LIN {X 0,Y 305.425,Z 148.042,A -85,B 0,C 180,E1 -16066.344,E2 -16066.344} C_VEL
LIN {X 0,Y 305.415,Z 148.066,A -85,B 0,C 180,E1 -16069.885,E2 -16069.885} C_VEL
LIN {X 0,Y 305.467,Z 148.054,A -85,B 0,C 180,E1 -16073.636,E2 -16073.636} C_VEL
LIN {X 0,Y 305.47,Z 148.051,A -85,B 0,C 180,E1 -16076.483,E2 -16076.483} C_VEL
LIN {X 0,Y 305.436,Z 148.065,A -85,B 0,C 180,E1 -16079.587,E2 -16079.587} C_VEL
LIN {X 0,Y 305.456,Z 148.059,A -85,B 0,C 180,E1 -16082.602,E2 -16082.602} C_VEL
LIN {X 0,Y 305.461,Z 148.064,A -85,B 0,C 180,E1 -16085.534,E2 -16085.534} C_VEL
LIN {X 0,Y 305.504,Z 148.057,A -85,B 0,C 180,E1 -16089.813,E2 -16089.813} C_VEL
LIN {X 0,Y 305.56,Z 148.153,A -85,B 0,C 180,E1 -16092.669,E2 -16092.669} C_VEL
LIN {X 0,Y 306.725,Z 151.141,A -85,B 0,C 180,E1 -16092.931,E2 -16092.931} C_VEL
LIN {X 0,Y 311.745,Z 160.729,A -85,B 0,C 180,E1 -16093.747,E2 -16093.747} C_VEL
LIN {X 0,Y 320.601,Z 180.222,A -85,B 0,C 180,E1 -16095.182,E2 -16095.182} C_VEL
LIN {X 0,Y 326.991,Z 195.626,A -85,B 0,C 180,E1 -16096.196,E2 -16096.196} C_VEL
LIN {X 0,Y 326.331,Z 222.308,A -85,B 0,C 180,E1 -16096.802,E2 -16096.802} C_VEL
LIN {X 0,Y 323.34,Z 313.108,A -85,B 0,C 180,E1 -16098.83,E2 -16098.83} C_VEL
LIN {X 0,Y 322.302,Z 328.917,A -85,B 0,C 180,E1 -16099.427,E2 -16099.427} C_VEL
LIN {X 0,Y 321.017,Z 343.579,A -85,B 0,C 180,E1 -16100.231,E2 -16100.231} C_VEL
LIN {X 0,Y 319.266,Z 358.274,A -85,B 0,C 180,E1 -16101.295,E2 -16101.295} C_VEL
LIN {X 0,Y 317.48,Z 371.58,A -85,B 0,C 180,E1 -16102.527,E2 -16102.527} C_VEL
LIN {X 0,Y 315.3,Z 385.197,A -85,B 0,C 180,E1 -16104.082,E2 -16104.082} C_VEL
LIN {X 0,Y 313.172,Z 397.517,A -85,B 0,C 180,E1 -16105.817,E2 -16105.817} C_VEL
LIN {X 0,Y 311.183,Z 408.729,A -85,B 0,C 180,E1 -16107.734,E2 -16107.734} C_VEL
LIN {X 0,Y 309.193,Z 419.649,A -85,B 0,C 180,E1 -16109.999,E2 -16109.999} C_VEL
LIN {X 0,Y 307.452,Z 428.742,A -85,B 0,C 180,E1 -16112.292,E2 -16112.292} C_VEL
LIN {X 0,Y 306.162,Z 436.275,A -85,B 0,C 180,E1 -16114.608,E2 -16114.608} C_VEL
LIN {X 0,Y 305.104,Z 442.962,A -85,B 0,C 180,E1 -16117.129,E2 -16117.129} C_VEL
LIN {X 0,Y 304.26,Z 448.88,A -85,B 0,C 180,E1 -16119.976,E2 -16119.976} C_VEL
LIN {X 0,Y 303.878,Z 452.134,A -85,B 0,C 180,E1 -16122.013,E2 -16122.013} C_VEL
LIN {X 0,Y 303.455,Z 455.372,A -85,B 0,C 180,E1 -16124.759,E2 -16124.759} C_VEL
LIN {X 0,Y 303.371,Z 457.353,A -85,B 0,C 180,E1 -16127.527,E2 -16127.527} C_VEL
LIN {X 0,Y 303.342,Z 458.075,A -85,B 0,C 180,E1 -16130.336,E2 -16130.336} C_VEL
LIN {X 0,Y 303.492,Z 457.871,A -85,B 0,C 180,E1 -16132.135,E2 -16132.135} C_VEL
LIN {X 0,Y 303.727,Z 456.748,A -85,B 0,C 180,E1 -16134.614,E2 -16134.614} C_VEL
LIN {X 0,Y 304.341,Z 454.188,A -85,B 0,C 180,E1 -16137.506,E2 -16137.506} C_VEL
LIN {X 0,Y 305.312,Z 450.177,A -85,B 0,C 180,E1 -16140.425,E2 -16140.425} C_VEL
LIN {X 0,Y 306.808,Z 444.597,A -85,B 0,C 180,E1 -16143.35,E2 -16143.35} C_VEL
LIN {X 0,Y 308.291,Z 439.231,A -85,B 0,C 180,E1 -16145.543,E2 -16145.543} C_VEL
LIN {X 0,Y 310.472,Z 431.577,A -85,B 0,C 180,E1 -16148.086,E2 -16148.086} C_VEL
LIN {X 0,Y 313.128,Z 422.138,A -85,B 0,C 180,E1 -16150.608,E2 -16150.608} C_VEL
LIN {X 0,Y 315.898,Z 412.215,A -85,B 0,C 180,E1 -16152.762,E2 -16152.762} C_VEL
LIN {X 0,Y 318.717,Z 401.62,A -85,B 0,C 180,E1 -16154.657,E2 -16154.657} C_VEL
LIN {X 0,Y 321.534,Z 389.978,A -85,B 0,C 180,E1 -16156.388,E2 -16156.388} C_VEL
LIN {X 0,Y 324.49,Z 376.91,A -85,B 0,C 180,E1 -16157.965,E2 -16157.965} C_VEL
LIN {X 0,Y 327.018,Z 363.873,A -85,B 0,C 180,E1 -16159.244,E2 -16159.244} C_VEL
LIN {X 0,Y 327.93,Z 358.533,A -85,B 0,C 180,E1 -16159.697,E2 -16159.697} C_VEL
LIN {X 0,Y 328.286,Z 353.289,A -85,B 0,C 180,E1 -16160.17,E2 -16160.17} C_VEL
LIN {X 0,Y 326.223,Z 337.898,A -85,B 0,C 180,E1 -16161.711,E2 -16161.711} C_VEL
LIN {X 0,Y 326.007,Z 332.452,A -85,B 0,C 180,E1 -16162.106,E2 -16162.106} C_VEL
LIN {X 0,Y 326.158,Z 330.579,A -85,B 0,C 180,E1 -16162.207,E2 -16162.207} C_VEL
LIN {X 0,Y 327.542,Z 315.801,A -85,B 0,C 180,E1 -16162.767,E2 -16162.767} C_VEL
LIN {X 0,Y 328.616,Z 292.672,A -85,B 0,C 180,E1 -16163.339,E2 -16163.339} C_VEL
LIN {X 0,Y 332.473,Z 206.469,A -85,B 0,C 180,E1 -16165.255,E2 -16165.255} C_VEL
LIN {X 0,Y 326.364,Z 194.052,A -85,B 0,C 180,E1 -16166.6,E2 -16166.6} C_VEL
LIN {X 0,Y 319.353,Z 181.411,A -85,B 0,C 180,E1 -16168.205,E2 -16168.205} C_VEL
LIN {X 0,Y 312.337,Z 169.916,A -85,B 0,C 180,E1 -16169.909,E2 -16169.909} C_VEL
LIN {X 0,Y 305.127,Z 159.284,A -85,B 0,C 180,E1 -16171.777,E2 -16171.777} C_VEL
LIN {X 0,Y 301.722,Z 154.601,A -85,B 0,C 180,E1 -16172.704,E2 -16172.704} C_VEL
LIN {X 0,Y 299.117,Z 151.181,A -85,B 0,C 180,E1 -16173.438,E2 -16173.438} C_VEL
LIN {X 0,Y 298.731,Z 150.191,A -85,B 0,C 180,E1 -16173.604,E2 -16173.604} C_VEL
LIN {X 0,Y 298.46,Z 148.929,A -85,B 0,C 180,E1 -16174.174,E2 -16174.174} C_VEL
LIN {X 0,Y 298.419,Z 148.934,A -85,B 0,C 180,E1 -16177.863,E2 -16177.863} C_VEL
LIN {X 0,Y 298.508,Z 148.928,A -85,B 0,C 180,E1 -16180.754,E2 -16180.754} C_VEL
LIN {X 0,Y 298.585,Z 148.91,A -85,B 0,C 180,E1 -16184.994,E2 -16184.994} C_VEL
LIN {X 0,Y 298.594,Z 148.914,A -85,B 0,C 180,E1 -16189.146,E2 -16189.146} C_VEL
LIN {X 0,Y 298.758,Z 148.89,A -85,B 0,C 180,E1 -16191.885,E2 -16191.885} C_VEL
LIN {X 0,Y 298.658,Z 148.898,A -85,B 0,C 180,E1 -16194.598,E2 -16194.598} C_VEL
LIN {X 0,Y 298.922,Z 148.868,A -85,B 0,C 180,E1 -16198.652,E2 -16198.652} C_VEL
LIN {X 0,Y 298.922,Z 148.866,A -85,B 0,C 180,E1 -16201.347,E2 -16201.347} C_VEL
LIN {X 0,Y 298.641,Z 148.901,A -85,B 0,C 180,E1 -16205.401,E2 -16205.401} C_VEL
LIN {X 0,Y 298.707,Z 148.892,A -85,B 0,C 180,E1 -16208.821,E2 -16208.821} C_VEL
LIN {X 0,Y 298.551,Z 148.917,A -85,B 0,C 180,E1 -16213.615,E2 -16213.615} C_VEL
LIN {X 0,Y 298.548,Z 148.912,A -85,B 0,C 180,E1 -16216.408,E2 -16216.408} C_VEL
LIN {X 0,Y 298.511,Z 148.916,A -85,B 0,C 180,E1 -16219.655,E2 -16219.655} C_VEL
LIN {X 0,Y 298.456,Z 148.927,A -85,B 0,C 180,E1 -16223.597,E2 -16223.597} C_VEL
LIN {X 0,Y 298.488,Z 148.922,A -85,B 0,C 180,E1 -16226.574,E2 -16226.574} C_VEL
LIN {X 0,Y 298.419,Z 148.931,A -85,B 0,C 180,E1 -16229.641,E2 -16229.641} C_VEL
LIN {X 0,Y 298.393,Z 148.936,A -85,B 0,C 180,E1 -16232.8,E2 -16232.8} C_VEL
LIN {X 0,Y 298.442,Z 148.931,A -85,B 0,C 180,E1 -16236.807,E2 -16236.807} C_VEL
LIN {X 0,Y 298.403,Z 148.951,A -85,B 0,C 180,E1 -16241.258,E2 -16241.258} C_VEL
LIN {X 0,Y 301.892,Z 159.125,A -85,B 0,C 180,E1 -16245.702,E2 -16245.702} C_VEL
LIN {X 0,Y 302.524,Z 160.987,A -85,B 0,C 180,E1 -16246.372,E2 -16246.372} C_VEL
LIN {X 0,Y 305.677,Z 165.771,A -85,B 0,C 180,E1 -16247.234,E2 -16247.234} C_VEL
LIN {X 0,Y 310.675,Z 173.836,A -85,B 0,C 180,E1 -16248.552,E2 -16248.552} C_VEL
LIN {X 0,Y 315.895,Z 182.441,A -85,B 0,C 180,E1 -16249.854,E2 -16249.854} C_VEL
LIN {X 0,Y 323.059,Z 195.628,A -85,B 0,C 180,E1 -16251.551,E2 -16251.551} C_VEL
LIN {X 0,Y 330.619,Z 211.498,A -85,B 0,C 180,E1 -16253.263,E2 -16253.263} C_VEL
LIN {X 0,Y 331.46,Z 214.963,A -85,B 0,C 180,E1 -16253.496,E2 -16253.496} C_VEL
LIN {X 0,Y 331.991,Z 218.821,A -85,B 0,C 180,E1 -16253.69,E2 -16253.69} C_VEL
LIN {X 0,Y 327.142,Z 328.832,A -85,B 0,C 180,E1 -16256.183,E2 -16256.183} C_VEL
LIN {X 0,Y 325.74,Z 343.604,A -85,B 0,C 180,E1 -16256.714,E2 -16256.714} C_VEL
LIN {X 0,Y 323.571,Z 358.814,A -85,B 0,C 180,E1 -16257.482,E2 -16257.482} C_VEL
LIN {X 0,Y 321.291,Z 372.892,A -85,B 0,C 180,E1 -16258.471,E2 -16258.471} C_VEL
LIN {X 0,Y 318.787,Z 385.068,A -85,B 0,C 180,E1 -16259.532,E2 -16259.532} C_VEL
LIN {X 0,Y 316.108,Z 397.601,A -85,B 0,C 180,E1 -16260.9,E2 -16260.9} C_VEL
LIN {X 0,Y 312.767,Z 410.359,A -85,B 0,C 180,E1 -16262.572,E2 -16262.572} C_VEL
LIN {X 0,Y 309.669,Z 421.95,A -85,B 0,C 180,E1 -16264.456,E2 -16264.456} C_VEL
LIN {X 0,Y 306.731,Z 431.991,A -85,B 0,C 180,E1 -16266.419,E2 -16266.419} C_VEL
LIN {X 0,Y 304.14,Z 441.389,A -85,B 0,C 180,E1 -16268.658,E2 -16268.658} C_VEL
LIN {X 0,Y 301.847,Z 449.475,A -85,B 0,C 180,E1 -16270.976,E2 -16270.976} C_VEL
LIN {X 0,Y 299.69,Z 457.055,A -85,B 0,C 180,E1 -16273.656,E2 -16273.656} C_VEL
LIN {X 0,Y 298.256,Z 463.123,A -85,B 0,C 180,E1 -16276.371,E2 -16276.371} C_VEL
LIN {X 0,Y 297.22,Z 467.814,A -85,B 0,C 180,E1 -16279.096,E2 -16279.096} C_VEL
LIN {X 0,Y 296.703,Z 471.255,A -85,B 0,C 180,E1 -16281.83,E2 -16281.83} C_VEL
LIN {X 0,Y 296.51,Z 473.52,A -85,B 0,C 180,E1 -16284.56,E2 -16284.56} C_VEL
LIN {X 0,Y 296.511,Z 474.65,A -85,B 0,C 180,E1 -16287.283,E2 -16287.283} C_VEL
LIN {X 0,Y 296.517,Z 474.641,A -85,B 0,C 180,E1 -16290.001,E2 -16290.001} C_VEL
LIN {X 0,Y 296.521,Z 473.418,A -85,B 0,C 180,E1 -16292.718,E2 -16292.718} C_VEL
LIN {X 0,Y 296.544,Z 470.934,A -85,B 0,C 180,E1 -16295.509,E2 -16295.509} C_VEL
LIN {X 0,Y 296.72,Z 467.357,A -85,B 0,C 180,E1 -16298.171,E2 -16298.171} C_VEL
LIN {X 0,Y 297.077,Z 462.361,A -85,B 0,C 180,E1 -16300.91,E2 -16300.91} C_VEL
LIN {X 0,Y 297.953,Z 455.897,A -85,B 0,C 180,E1 -16303.644,E2 -16303.644} C_VEL
LIN {X 0,Y 299.002,Z 449.017,A -85,B 0,C 180,E1 -16305.998,E2 -16305.998} C_VEL
LIN {X 0,Y 300.499,Z 440.454,A -85,B 0,C 180,E1 -16308.406,E2 -16308.406} C_VEL
LIN {X 0,Y 302.506,Z 430.248,A -85,B 0,C 180,E1 -16310.751,E2 -16310.751} C_VEL
LIN {X 0,Y 304.47,Z 419.22,A -85,B 0,C 180,E1 -16312.848,E2 -16312.848} C_VEL
LIN {X 0,Y 306.71,Z 407.241,A -85,B 0,C 180,E1 -16314.721,E2 -16314.721} C_VEL
LIN {X 0,Y 308.879,Z 394.65,A -85,B 0,C 180,E1 -16316.34,E2 -16316.34} C_VEL
LIN {X 0,Y 311.197,Z 380.874,A -85,B 0,C 180,E1 -16317.762,E2 -16317.762} C_VEL
LIN {X 0,Y 313.007,Z 367.492,A -85,B 0,C 180,E1 -16318.876,E2 -16318.876} C_VEL
LIN {X 0,Y 314.765,Z 351.771,A -85,B 0,C 180,E1 -16319.881,E2 -16319.881} C_VEL
LIN {X 0,Y 316.114,Z 336.594,A -85,B 0,C 180,E1 -16320.569,E2 -16320.569} C_VEL
LIN {X 0,Y 316.964,Z 320.811,A -85,B 0,C 180,E1 -16321.033,E2 -16321.033} C_VEL
LIN {X 0,Y 320.409,Z 215.479,A -85,B 0,C 180,E1 -16323.398,E2 -16323.398} C_VEL
LIN {X 0,Y 317.55,Z 198.45,A -85,B 0,C 180,E1 -16324.12,E2 -16324.12} C_VEL
LIN {X 0,Y 308.738,Z 177.194,A -85,B 0,C 180,E1 -16325.6,E2 -16325.6} C_VEL
LIN {X 0,Y 301.978,Z 162.23,A -85,B 0,C 180,E1 -16326.8,E2 -16326.8} C_VEL
LIN {X 0,Y 298.869,Z 150.636,A -85,B 0,C 180,E1 -16330.161,E2 -16330.161} C_VEL
LIN {X 0,Y 298.418,Z 148.94,A -85,B 0,C 180,E1 -16330.712,E2 -16330.712} C_VEL
LIN {X 0,Y 298.4,Z 148.942,A -85,B 0,C 180,E1 -16333.104,E2 -16333.104} C_VEL
LIN {X 0,Y 298.404,Z 148.945,A -85,B 0,C 180,E1 -16336.922,E2 -16336.922} C_VEL
LIN {X 0,Y 298.401,Z 148.929,A -85,B 0,C 180,E1 -16341.008,E2 -16341.008} C_VEL
LIN {X 0,Y 298.42,Z 148.935,A -85,B 0,C 180,E1 -16343.931,E2 -16343.931} C_VEL
LIN {X 0,Y 298.391,Z 148.939,A -85,B 0,C 180,E1 -16347.986,E2 -16347.986} C_VEL
LIN {X 0,Y 298.415,Z 148.91,A -85,B 0,C 180,E1 -16351.9,E2 -16351.9} C_VEL
LIN {X 0,Y 298.443,Z 148.927,A -85,B 0,C 180,E1 -16354.921,E2 -16354.921} C_VEL
LIN {X 0,Y 298.418,Z 148.93,A -85,B 0,C 180,E1 -16357.864,E2 -16357.864} C_VEL
LIN {X 0,Y 298.509,Z 148.928,A -85,B 0,C 180,E1 -16360.755,E2 -16360.755} C_VEL
LIN {X 0,Y 298.589,Z 148.918,A -85,B 0,C 180,E1 -16364.995,E2 -16364.995} C_VEL
LIN {X 0,Y 298.587,Z 148.916,A -85,B 0,C 180,E1 -16369.147,E2 -16369.147} C_VEL
LIN {X 0,Y 298.702,Z 148.897,A -85,B 0,C 180,E1 -16371.885,E2 -16371.885} C_VEL
LIN {X 0,Y 298.632,Z 148.912,A -85,B 0,C 180,E1 -16374.599,E2 -16374.599} C_VEL
LIN {X 0,Y 298.907,Z 148.844,A -85,B 0,C 180,E1 -16378.653,E2 -16378.653} C_VEL
LIN {X 0,Y 298.906,Z 148.857,A -85,B 0,C 180,E1 -16381.348,E2 -16381.348} C_VEL
LIN {X 0,Y 298.739,Z 148.886,A -85,B 0,C 180,E1 -16386.756,E2 -16386.756} C_VEL
LIN {X 0,Y 298.628,Z 148.873,A -85,B 0,C 180,E1 -16389.483,E2 -16389.483} C_VEL
LIN {X 0,Y 298.512,Z 148.922,A -85,B 0,C 180,E1 -16393.618,E2 -16393.618} C_VEL
LIN {X 0,Y 298.431,Z 148.927,A -85,B 0,C 180,E1 -16396.416,E2 -16396.416} C_VEL
LIN {X 0,Y 298.427,Z 148.939,A -85,B 0,C 180,E1 -16399.606,E2 -16399.606} C_VEL
LIN {X 0,Y 298.385,Z 148.94,A -85,B 0,C 180,E1 -16403.604,E2 -16403.604} C_VEL
LIN {X 0,Y 298.405,Z 148.933,A -85,B 0,C 180,E1 -16406.583,E2 -16406.583} C_VEL
LIN {X 0,Y 298.36,Z 148.911,A -85,B 0,C 180,E1 -16409.648,E2 -16409.648} C_VEL
LIN {X 0,Y 298.397,Z 148.934,A -85,B 0,C 180,E1 -16412.801,E2 -16412.801} C_VEL
LIN {X 0,Y 298.43,Z 148.915,A -85,B 0,C 180,E1 -16416.802,E2 -16416.802} C_VEL
LIN {X 0,Y 298.379,Z 148.92,A -85,B 0,C 180,E1 -16419.492,E2 -16419.492} C_VEL
LIN {X 0,Y 298.375,Z 148.94,A -85,B 0,C 180,E1 -16423.097,E2 -16423.097} C_VEL
LIN {X 0,Y 298.375,Z 148.925,A -85,B 0,C 180,E1 -16426.915,E2 -16426.915} C_VEL
LIN {X 0,Y 298.356,Z 148.935,A -85,B 0,C 180,E1 -16431.019,E2 -16431.019} C_VEL
LIN {X 0,Y 298.41,Z 148.934,A -85,B 0,C 180,E1 -16433.928,E2 -16433.928} C_VEL
LIN {X 0,Y 298.398,Z 148.927,A -85,B 0,C 180,E1 -16437.199,E2 -16437.199} C_VEL
LIN {X 0,Y 298.407,Z 148.937,A -85,B 0,C 180,E1 -16440.625,E2 -16440.625} C_VEL
LIN {X 0,Y 298.427,Z 148.94,A -85,B 0,C 180,E1 -16444.918,E2 -16444.918} C_VEL
LIN {X 0,Y 298.409,Z 148.94,A -85,B 0,C 180,E1 -16447.862,E2 -16447.862} C_VEL
LIN {X 0,Y 298.507,Z 148.905,A -85,B 0,C 180,E1 -16451.911,E2 -16451.911} C_VEL
LIN {X 0,Y 299.447,Z 151.652,A -85,B 0,C 180,E1 -16452.105,E2 -16452.105} C_VEL
LIN {X 0,Y 304.331,Z 160.351,A -85,B 0,C 180,E1 -16452.914,E2 -16452.914} C_VEL
LIN {X 0,Y 312.231,Z 177.22,A -85,B 0,C 180,E1 -16454.24,E2 -16454.24} C_VEL
LIN {X 0,Y 320.714,Z 197.388,A -85,B 0,C 180,E1 -16455.636,E2 -16455.636} C_VEL
LIN {X 0,Y 320.022,Z 223.664,A -85,B 0,C 180,E1 -16456.242,E2 -16456.242} C_VEL
LIN {X 0,Y 316.94,Z 313.47,A -85,B 0,C 180,E1 -16458.285,E2 -16458.285} C_VEL
LIN {X 0,Y 315.891,Z 328.921,A -85,B 0,C 180,E1 -16458.877,E2 -16458.877} C_VEL
LIN {X 0,Y 314.556,Z 343.739,A -85,B 0,C 180,E1 -16459.703,E2 -16459.703} C_VEL
LIN {X 0,Y 312.76,Z 358.435,A -85,B 0,C 180,E1 -16460.786,E2 -16460.786} C_VEL
LIN {X 0,Y 310.904,Z 371.752,A -85,B 0,C 180,E1 -16462.041,E2 -16462.041} C_VEL
LIN {X 0,Y 308.646,Z 385.376,A -85,B 0,C 180,E1 -16463.626,E2 -16463.626} C_VEL
LIN {X 0,Y 306.47,Z 397.7,A -85,B 0,C 180,E1 -16465.396,E2 -16465.396} C_VEL
LIN {X 0,Y 304.389,Z 408.93,A -85,B 0,C 180,E1 -16467.353,E2 -16467.353} C_VEL
LIN {X 0,Y 302.483,Z 419.016,A -85,B 0,C 180,E1 -16469.474,E2 -16469.474} C_VEL
LIN {X 0,Y 300.528,Z 428.952,A -85,B 0,C 180,E1 -16472.01,E2 -16472.01} C_VEL
LIN {X 0,Y 299.323,Z 435.475,A -85,B 0,C 180,E1 -16474.039,E2 -16474.039} C_VEL
LIN {X 0,Y 298.142,Z 442.725,A -85,B 0,C 180,E1 -16476.768,E2 -16476.768} C_VEL
LIN {X 0,Y 297.272,Z 448.457,A -85,B 0,C 180,E1 -16479.525,E2 -16479.525} C_VEL
LIN {X 0,Y 296.709,Z 452.807,A -85,B 0,C 180,E1 -16482.308,E2 -16482.308} C_VEL
LIN {X 0,Y 296.334,Z 455.872,A -85,B 0,C 180,E1 -16485.122,E2 -16485.122} C_VEL
LIN {X 0,Y 296.286,Z 457.688,A -85,B 0,C 180,E1 -16487.96,E2 -16487.96} C_VEL
LIN {X 0,Y 296.279,Z 458.268,A -85,B 0,C 180,E1 -16490.843,E2 -16490.843} C_VEL
LIN {X 0,Y 296.514,Z 457.57,A -85,B 0,C 180,E1 -16493.761,E2 -16493.761} C_VEL
LIN {X 0,Y 297.054,Z 455.537,A -85,B 0,C 180,E1 -16496.712,E2 -16496.712} C_VEL
LIN {X 0,Y 297.943,Z 452.083,A -85,B 0,C 180,E1 -16499.693,E2 -16499.693} C_VEL
LIN {X 0,Y 299.319,Z 447.098,A -85,B 0,C 180,E1 -16502.686,E2 -16502.686} C_VEL
LIN {X 0,Y 300.937,Z 441.641,A -85,B 0,C 180,E1 -16505.175,E2 -16505.175} C_VEL
LIN {X 0,Y 302.879,Z 435.069,A -85,B 0,C 180,E1 -16507.591,E2 -16507.591} C_VEL
LIN {X 0,Y 305.412,Z 426.604,A -85,B 0,C 180,E1 -16510.115,E2 -16510.115} C_VEL
LIN {X 0,Y 308.078,Z 417.654,A -85,B 0,C 180,E1 -16512.296,E2 -16512.296} C_VEL
LIN {X 0,Y 311.156,Z 406.943,A -85,B 0,C 180,E1 -16514.442,E2 -16514.442} C_VEL
LIN {X 0,Y 314.202,Z 395.585,A -85,B 0,C 180,E1 -16516.308,E2 -16516.308} C_VEL
LIN {X 0,Y 317.152,Z 383.564,A -85,B 0,C 180,E1 -16517.931,E2 -16517.931} C_VEL
LIN {X 0,Y 319.857,Z 371.29,A -85,B 0,C 180,E1 -16519.292,E2 -16519.292} C_VEL
LIN {X 0,Y 322.294,Z 357.979,A -85,B 0,C 180,E1 -16520.499,E2 -16520.499} C_VEL
LIN {X 0,Y 324.503,Z 344.079,A -85,B 0,C 180,E1 -16521.479,E2 -16521.479} C_VEL
LIN {X 0,Y 326.158,Z 330.579,A -85,B 0,C 180,E1 -16522.207,E2 -16522.207} C_VEL
LIN {X 0,Y 326.261,Z 324.959,A -85,B 0,C 180,E1 -16522.528,E2 -16522.528} C_VEL
LIN {X 0,Y 323.394,Z 308.503,A -85,B 0,C 180,E1 -16523.642,E2 -16523.642} C_VEL
LIN {X 0,Y 322.862,Z 302.795,A -85,B 0,C 180,E1 -16523.9,E2 -16523.9} C_VEL
LIN {X 0,Y 322.871,Z 300.849,A -85,B 0,C 180,E1 -16523.955,E2 -16523.955} C_VEL
LIN {X 0,Y 327.076,Z 208.883,A -85,B 0,C 180,E1 -16526.035,E2 -16526.035} C_VEL
LIN {X 0,Y 320.687,Z 195.996,A -85,B 0,C 180,E1 -16527.503,E2 -16527.503} C_VEL
LIN {X 0,Y 314.788,Z 185.399,A -85,B 0,C 180,E1 -16528.915,E2 -16528.915} C_VEL
LIN {X 0,Y 308.259,Z 174.605,A -85,B 0,C 180,E1 -16530.569,E2 -16530.569} C_VEL
LIN {X 0,Y 301.506,Z 164.511,A -85,B 0,C 180,E1 -16532.384,E2 -16532.384} C_VEL
LIN {X 0,Y 297.592,Z 159.111,A -85,B 0,C 180,E1 -16533.495,E2 -16533.495} C_VEL
LIN {X 0,Y 295.398,Z 155.951,A -85,B 0,C 180,E1 -16534.154,E2 -16534.154} C_VEL
LIN {X 0,Y 293.762,Z 154.239,A -85,B 0,C 180,E1 -16534.634,E2 -16534.634} C_VEL
LIN {X 0,Y 291.995,Z 151.912,A -85,B 0,C 180,E1 -16535.184,E2 -16535.184} C_VEL
LIN {X 0,Y 291.497,Z 150.493,A -85,B 0,C 180,E1 -16535.423,E2 -16535.423} C_VEL
LIN {X 0,Y 291.366,Z 149.793,A -85,B 0,C 180,E1 -16535.791,E2 -16535.791} C_VEL
LIN {X 0,Y 291.458,Z 149.802,A -85,B 0,C 180,E1 -16540.269,E2 -16540.269} C_VEL
LIN {X 0,Y 291.514,Z 149.792,A -85,B 0,C 180,E1 -16544.652,E2 -16544.652} C_VEL
LIN {X 0,Y 291.537,Z 149.791,A -85,B 0,C 180,E1 -16548.88,E2 -16548.88} C_VEL
LIN {X 0,Y 291.709,Z 149.766,A -85,B 0,C 180,E1 -16551.688,E2 -16551.688} C_VEL
LIN {X 0,Y 291.629,Z 149.774,A -85,B 0,C 180,E1 -16554.468,E2 -16554.468} C_VEL
LIN {X 0,Y 291.888,Z 149.743,A -85,B 0,C 180,E1 -16558.62,E2 -16558.62} C_VEL
LIN {X 0,Y 291.888,Z 149.742,A -85,B 0,C 180,E1 -16561.379,E2 -16561.379} C_VEL
LIN {X 0,Y 291.609,Z 149.777,A -85,B 0,C 180,E1 -16565.532,E2 -16565.532} C_VEL
LIN {X 0,Y 291.667,Z 149.769,A -85,B 0,C 180,E1 -16568.911,E2 -16568.911} C_VEL
LIN {X 0,Y 291.517,Z 149.787,A -85,B 0,C 180,E1 -16572.531,E2 -16572.531} C_VEL
LIN {X 0,Y 291.554,Z 149.786,A -85,B 0,C 180,E1 -16575.376,E2 -16575.376} C_VEL
LIN {X 0,Y 291.449,Z 149.796,A -85,B 0,C 180,E1 -16579.874,E2 -16579.874} C_VEL
LIN {X 0,Y 291.399,Z 149.811,A -85,B 0,C 180,E1 -16584.205,E2 -16584.205} C_VEL
LIN {X 0,Y 291.421,Z 149.807,A -85,B 0,C 180,E1 -16587.271,E2 -16587.271} C_VEL
LIN {X 0,Y 291.336,Z 149.819,A -85,B 0,C 180,E1 -16590.436,E2 -16590.436} C_VEL
LIN {X 0,Y 291.342,Z 149.821,A -85,B 0,C 180,E1 -16593.698,E2 -16593.698} C_VEL
LIN {X 0,Y 291.37,Z 149.803,A -85,B 0,C 180,E1 -16597.253,E2 -16597.253} C_VEL
LIN {X 0,Y 291.357,Z 149.822,A -85,B 0,C 180,E1 -16599.678,E2 -16599.678} C_VEL
LIN {X 0,Y 293.734,Z 156.797,A -85,B 0,C 180,E1 -16602.992,E2 -16602.992} C_VEL
LIN {X 0,Y 295.134,Z 160.601,A -85,B 0,C 180,E1 -16604.625,E2 -16604.625} C_VEL
LIN {X 0,Y 298.393,Z 165.535,A -85,B 0,C 180,E1 -16605.601,E2 -16605.601} C_VEL
LIN {X 0,Y 303.702,Z 173.755,A -85,B 0,C 180,E1 -16607.098,E2 -16607.098} C_VEL
LIN {X 0,Y 307.066,Z 179.192,A -85,B 0,C 180,E1 -16608.004,E2 -16608.004} C_VEL
LIN {X 0,Y 312.288,Z 188.018,A -85,B 0,C 180,E1 -16609.355,E2 -16609.355} C_VEL
LIN {X 0,Y 319.016,Z 200.662,A -85,B 0,C 180,E1 -16611.009,E2 -16611.009} C_VEL
LIN {X 0,Y 326.015,Z 215.704,A -85,B 0,C 180,E1 -16612.657,E2 -16612.657} C_VEL
LIN {X 0,Y 326.688,Z 219.828,A -85,B 0,C 180,E1 -16612.889,E2 -16612.889} C_VEL
LIN {X 0,Y 321.672,Z 328.58,A -85,B 0,C 180,E1 -16615.386,E2 -16615.386} C_VEL
LIN {X 0,Y 320.189,Z 343.354,A -85,B 0,C 180,E1 -16615.917,E2 -16615.917} C_VEL
LIN {X 0,Y 317.872,Z 359.13,A -85,B 0,C 180,E1 -16616.73,E2 -16616.73} C_VEL
LIN {X 0,Y 315.324,Z 374.007,A -85,B 0,C 180,E1 -16617.805,E2 -16617.805} C_VEL
LIN {X 0,Y 312.435,Z 387.504,A -85,B 0,C 180,E1 -16619.033,E2 -16619.033} C_VEL
LIN {X 0,Y 309.303,Z 400.837,A -85,B 0,C 180,E1 -16620.57,E2 -16620.57} C_VEL
LIN {X 0,Y 305.979,Z 413.019,A -85,B 0,C 180,E1 -16622.282,E2 -16622.282} C_VEL
LIN {X 0,Y 302.787,Z 424.147,A -85,B 0,C 180,E1 -16624.202,E2 -16624.202} C_VEL
LIN {X 0,Y 299.509,Z 435.022,A -85,B 0,C 180,E1 -16626.491,E2 -16626.491} C_VEL
LIN {X 0,Y 296.761,Z 444.069,A -85,B 0,C 180,E1 -16628.829,E2 -16628.829} C_VEL
LIN {X 0,Y 294.496,Z 451.625,A -85,B 0,C 180,E1 -16631.206,E2 -16631.206} C_VEL
LIN {X 0,Y 292.369,Z 458.57,A -85,B 0,C 180,E1 -16633.879,E2 -16633.879} C_VEL
LIN {X 0,Y 291.002,Z 464.385,A -85,B 0,C 180,E1 -16636.737,E2 -16636.737} C_VEL
LIN {X 0,Y 290.193,Z 467.789,A -85,B 0,C 180,E1 -16638.829,E2 -16638.829} C_VEL
LIN {X 0,Y 289.627,Z 471.174,A -85,B 0,C 180,E1 -16641.629,E2 -16641.629} C_VEL
LIN {X 0,Y 289.425,Z 473.495,A -85,B 0,C 180,E1 -16644.612,E2 -16644.612} C_VEL
LIN {X 0,Y 289.414,Z 474.463,A -85,B 0,C 180,E1 -16647.217,E2 -16647.217} C_VEL
LIN {X 0,Y 289.434,Z 474.41,A -85,B 0,C 180,E1 -16650.001,E2 -16650.001} C_VEL
LIN {X 0,Y 289.447,Z 473.156,A -85,B 0,C 180,E1 -16652.784,E2 -16652.784} C_VEL
LIN {X 0,Y 289.474,Z 470.694,A -85,B 0,C 180,E1 -16655.574,E2 -16655.574} C_VEL
LIN {X 0,Y 289.635,Z 466.985,A -85,B 0,C 180,E1 -16658.372,E2 -16658.372} C_VEL
LIN {X 0,Y 290.043,Z 461.928,A -85,B 0,C 180,E1 -16661.178,E2 -16661.178} C_VEL
LIN {X 0,Y 290.98,Z 455.395,A -85,B 0,C 180,E1 -16663.977,E2 -16663.977} C_VEL
LIN {X 0,Y 292.321,Z 447.186,A -85,B 0,C 180,E1 -16666.769,E2 -16666.769} C_VEL
LIN {X 0,Y 293.914,Z 438.405,A -85,B 0,C 180,E1 -16669.196,E2 -16669.196} C_VEL
LIN {X 0,Y 295.759,Z 429.484,A -85,B 0,C 180,E1 -16671.247,E2 -16671.247} C_VEL
LIN {X 0,Y 297.805,Z 418.622,A -85,B 0,C 180,E1 -16673.339,E2 -16673.339} C_VEL
LIN {X 0,Y 300.189,Z 406.232,A -85,B 0,C 180,E1 -16675.295,E2 -16675.295} C_VEL
LIN {X 0,Y 302.43,Z 393.466,A -85,B 0,C 180,E1 -16676.947,E2 -16676.947} C_VEL
LIN {X 0,Y 304.827,Z 379.454,A -85,B 0,C 180,E1 -16678.394,E2 -16678.394} C_VEL
LIN {X 0,Y 306.818,Z 365.062,A -85,B 0,C 180,E1 -16679.577,E2 -16679.577} C_VEL
LIN {X 0,Y 308.494,Z 350.26,A -85,B 0,C 180,E1 -16680.505,E2 -16680.505} C_VEL
LIN {X 0,Y 309.807,Z 335.59,A -85,B 0,C 180,E1 -16681.166,E2 -16681.166} C_VEL
LIN {X 0,Y 310.657,Z 319.334,A -85,B 0,C 180,E1 -16681.64,E2 -16681.64} C_VEL
LIN {X 0,Y 314.088,Z 215.808,A -85,B 0,C 180,E1 -16684.015,E2 -16684.015} C_VEL
LIN {X 0,Y 311.595,Z 201.047,A -85,B 0,C 180,E1 -16684.66,E2 -16684.66} C_VEL
LIN {X 0,Y 302.996,Z 180.293,A -85,B 0,C 180,E1 -16686.151,E2 -16686.151} C_VEL
LIN {X 0,Y 295.768,Z 164.685,A -85,B 0,C 180,E1 -16687.437,E2 -16687.437} C_VEL
LIN {X 0,Y 294.682,Z 162.011,A -85,B 0,C 180,E1 -16687.675,E2 -16687.675} C_VEL
LIN {X 0,Y 291.334,Z 149.821,A -85,B 0,C 180,E1 -16691.358,E2 -16691.358} C_VEL
LIN {X 0,Y 291.291,Z 149.83,A -85,B 0,C 180,E1 -16695.599,E2 -16695.599} C_VEL
LIN {X 0,Y 291.334,Z 149.821,A -85,B 0,C 180,E1 -16699.358,E2 -16699.358} C_VEL
LIN {X 0,Y 291.406,Z 149.811,A -85,B 0,C 180,E1 -16702.92,E2 -16702.92} C_VEL
LIN {X 0,Y 291.346,Z 149.818,A -85,B 0,C 180,E1 -16706.302,E2 -16706.302} C_VEL
LIN {X 0,Y 291.367,Z 149.808,A -85,B 0,C 180,E1 -16710.269,E2 -16710.269} C_VEL
LIN {X 0,Y 291.362,Z 149.804,A -85,B 0,C 180,E1 -16714.267,E2 -16714.267} C_VEL
LIN {X 0,Y 291.373,Z 149.809,A -85,B 0,C 180,E1 -16717.299,E2 -16717.299} C_VEL
LIN {X 0,Y 291.443,Z 149.804,A -85,B 0,C 180,E1 -16720.27,E2 -16720.27} C_VEL
LIN {X 0,Y 291.501,Z 149.797,A -85,B 0,C 180,E1 -16724.666,E2 -16724.666} C_VEL
LIN {X 0,Y 291.533,Z 149.794,A -85,B 0,C 180,E1 -16728.881,E2 -16728.881} C_VEL
LIN {X 0,Y 291.655,Z 149.776,A -85,B 0,C 180,E1 -16731.687,E2 -16731.687} C_VEL
LIN {X 0,Y 291.602,Z 149.788,A -85,B 0,C 180,E1 -16734.468,E2 -16734.468} C_VEL
LIN {X 0,Y 291.875,Z 149.72,A -85,B 0,C 180,E1 -16738.621,E2 -16738.621} C_VEL
LIN {X 0,Y 291.873,Z 149.733,A -85,B 0,C 180,E1 -16741.38,E2 -16741.38} C_VEL
LIN {X 0,Y 291.691,Z 149.763,A -85,B 0,C 180,E1 -16746.92,E2 -16746.92} C_VEL
LIN {X 0,Y 291.571,Z 149.751,A -85,B 0,C 180,E1 -16749.714,E2 -16749.714} C_VEL
LIN {X 0,Y 291.475,Z 149.802,A -85,B 0,C 180,E1 -16753.953,E2 -16753.953} C_VEL
LIN {X 0,Y 291.383,Z 149.805,A -85,B 0,C 180,E1 -16756.825,E2 -16756.825} C_VEL
LIN {X 0,Y 291.368,Z 149.816,A -85,B 0,C 180,E1 -16759.827,E2 -16759.827} C_VEL
LIN {X 0,Y 291.329,Z 149.82,A -85,B 0,C 180,E1 -16764.212,E2 -16764.212} C_VEL
LIN {X 0,Y 291.332,Z 149.803,A -85,B 0,C 180,E1 -16767.281,E2 -16767.281} C_VEL
LIN {X 0,Y 291.305,Z 149.794,A -85,B 0,C 180,E1 -16770.441,E2 -16770.441} C_VEL
LIN {X 0,Y 291.348,Z 149.817,A -85,B 0,C 180,E1 -16773.699,E2 -16773.699} C_VEL
LIN {X 0,Y 291.357,Z 149.79,A -85,B 0,C 180,E1 -16777.248,E2 -16777.248} C_VEL
LIN {X 0,Y 291.305,Z 149.814,A -85,B 0,C 180,E1 -16780.648,E2 -16780.648} C_VEL
LIN {X 0,Y 291.287,Z 149.811,A -85,B 0,C 180,E1 -16784.404,E2 -16784.404} C_VEL
LIN {X 0,Y 291.3,Z 149.821,A -85,B 0,C 180,E1 -16788.411,E2 -16788.411} C_VEL
LIN {X 0,Y 291.391,Z 149.798,A -85,B 0,C 180,E1 -16792.916,E2 -16792.916} C_VEL
LIN {X 0,Y 291.349,Z 149.811,A -85,B 0,C 180,E1 -16796.301,E2 -16796.301} C_VEL
LIN {X 0,Y 291.37,Z 149.817,A -85,B 0,C 180,E1 -16800.268,E2 -16800.268} C_VEL
LIN {X 0,Y 291.352,Z 149.822,A -85,B 0,C 180,E1 -16804.265,E2 -16804.265} C_VEL
LIN {X 0,Y 291.365,Z 149.819,A -85,B 0,C 180,E1 -16807.298,E2 -16807.298} C_VEL
LIN {X 0,Y 291.456,Z 149.79,A -85,B 0,C 180,E1 -16811.068,E2 -16811.068} C_VEL
LIN {X 0,Y 292.504,Z 152.718,A -85,B 0,C 180,E1 -16811.288,E2 -16811.288} C_VEL
LIN {X 0,Y 294.162,Z 155.518,A -85,B 0,C 180,E1 -16811.576,E2 -16811.576} C_VEL
LIN {X 0,Y 299.213,Z 164.669,A -85,B 0,C 180,E1 -16812.445,E2 -16812.445} C_VEL
LIN {X 0,Y 306.865,Z 181.158,A -85,B 0,C 180,E1 -16813.771,E2 -16813.771} C_VEL
LIN {X 0,Y 314.564,Z 199.511,A -85,B 0,C 180,E1 -16815.072,E2 -16815.072} C_VEL
LIN {X 0,Y 310.591,Z 313.59,A -85,B 0,C 180,E1 -16817.71,E2 -16817.71} C_VEL
LIN {X 0,Y 309.451,Z 329.633,A -85,B 0,C 180,E1 -16818.341,E2 -16818.341} C_VEL
LIN {X 0,Y 308.187,Z 343.239,A -85,B 0,C 180,E1 -16819.111,E2 -16819.111} C_VEL
LIN {X 0,Y 306.37,Z 358.025,A -85,B 0,C 180,E1 -16820.209,E2 -16820.209} C_VEL
LIN {X 0,Y 304.361,Z 371.919,A -85,B 0,C 180,E1 -16821.534,E2 -16821.534} C_VEL
LIN {X 0,Y 302.028,Z 385.55,A -85,B 0,C 180,E1 -16823.15,E2 -16823.15} C_VEL
LIN {X 0,Y 299.757,Z 397.884,A -85,B 0,C 180,E1 -16824.955,E2 -16824.955} C_VEL
LIN {X 0,Y 297.614,Z 409.112,A -85,B 0,C 180,E1 -16826.954,E2 -16826.954} C_VEL
LIN {X 0,Y 295.464,Z 420.006,A -85,B 0,C 180,E1 -16829.308,E2 -16829.308} C_VEL
LIN {X 0,Y 293.591,Z 429.144,A -85,B 0,C 180,E1 -16831.714,E2 -16831.714} C_VEL
LIN {X 0,Y 292.152,Z 436.688,A -85,B 0,C 180,E1 -16834.138,E2 -16834.138} C_VEL
LIN {X 0,Y 290.994,Z 443.737,A -85,B 0,C 180,E1 -16836.935,E2 -16836.935} C_VEL
LIN {X 0,Y 290.115,Z 449.291,A -85,B 0,C 180,E1 -16839.763,E2 -16839.763} C_VEL
LIN {X 0,Y 289.543,Z 453.47,A -85,B 0,C 180,E1 -16842.618,E2 -16842.618} C_VEL
LIN {X 0,Y 289.22,Z 456.367,A -85,B 0,C 180,E1 -16845.503,E2 -16845.503} C_VEL
LIN {X 0,Y 289.162,Z 458.076,A -85,B 0,C 180,E1 -16848.577,E2 -16848.577} C_VEL
LIN {X 0,Y 289.214,Z 458.432,A -85,B 0,C 180,E1 -16851.377,E2 -16851.377} C_VEL
LIN {X 0,Y 289.511,Z 457.563,A -85,B 0,C 180,E1 -16854.373,E2 -16854.373} C_VEL
LIN {X 0,Y 290.125,Z 455.356,A -85,B 0,C 180,E1 -16857.403,E2 -16857.403} C_VEL
LIN {X 0,Y 291.153,Z 451.715,A -85,B 0,C 180,E1 -16860.458,E2 -16860.458} C_VEL
LIN {X 0,Y 292.708,Z 446.521,A -85,B 0,C 180,E1 -16863.52,E2 -16863.52} C_VEL
LIN {X 0,Y 294.489,Z 440.929,A -85,B 0,C 180,E1 -16866.06,E2 -16866.06} C_VEL
LIN {X 0,Y 296.713,Z 433.984,A -85,B 0,C 180,E1 -16868.587,E2 -16868.587} C_VEL
LIN {X 0,Y 299.388,Z 425.474,A -85,B 0,C 180,E1 -16871.093,E2 -16871.093} C_VEL
LIN {X 0,Y 302.251,Z 416.246,A -85,B 0,C 180,E1 -16873.309,E2 -16873.309} C_VEL
LIN {X 0,Y 305.548,Z 405.212,A -85,B 0,C 180,E1 -16875.482,E2 -16875.482} C_VEL
LIN {X 0,Y 308.583,Z 394.181,A -85,B 0,C 180,E1 -16877.264,E2 -16877.264} C_VEL
LIN {X 0,Y 311.625,Z 382.137,A -85,B 0,C 180,E1 -16878.867,E2 -16878.867} C_VEL
LIN {X 0,Y 314.402,Z 369.812,A -85,B 0,C 180,E1 -16880.21,E2 -16880.21} C_VEL
LIN {X 0,Y 316.824,Z 357.031,A -85,B 0,C 180,E1 -16881.353,E2 -16881.353} C_VEL
LIN {X 0,Y 319.02,Z 343.493,A -85,B 0,C 180,E1 -16882.304,E2 -16882.304} C_VEL
LIN {X 0,Y 320.754,Z 329.833,A -85,B 0,C 180,E1 -16883.04,E2 -16883.04} C_VEL
LIN {X 0,Y 322.19,Z 314.435,A -85,B 0,C 180,E1 -16883.614,E2 -16883.614} C_VEL
LIN {X 0,Y 322.871,Z 300.849,A -85,B 0,C 180,E1 -16883.955,E2 -16883.955} C_VEL
LIN {X 0,Y 322.584,Z 295.062,A -85,B 0,C 180,E1 -16884.17,E2 -16884.17} C_VEL
LIN {X 0,Y 319.072,Z 276.536,A -85,B 0,C 180,E1 -16885.277,E2 -16885.277} C_VEL
LIN {X 0,Y 318.921,Z 270.746,A -85,B 0,C 180,E1 -16885.478,E2 -16885.478} C_VEL
LIN {X 0,Y 321.813,Z 211.794,A -85,B 0,C 180,E1 -16886.815,E2 -16886.815} C_VEL
LIN {X 0,Y 318.475,Z 204.507,A -85,B 0,C 180,E1 -16887.623,E2 -16887.623} C_VEL
LIN {X 0,Y 311.423,Z 191.299,A -85,B 0,C 180,E1 -16889.36,E2 -16889.36} C_VEL
LIN {X 0,Y 304.426,Z 179.563,A -85,B 0,C 180,E1 -16891.194,E2 -16891.194} C_VEL
LIN {X 0,Y 297.97,Z 169.82,A -85,B 0,C 180,E1 -16892.996,E2 -16892.996} C_VEL
LIN {X 0,Y 294.325,Z 164.726,A -85,B 0,C 180,E1 -16894.069,E2 -16894.069} C_VEL
LIN {X 0,Y 291.492,Z 160.789,A -85,B 0,C 180,E1 -16894.947,E2 -16894.947} C_VEL
LIN {X 0,Y 289.015,Z 157.873,A -85,B 0,C 180,E1 -16895.722,E2 -16895.722} C_VEL
LIN {X 0,Y 288.06,Z 156.041,A -85,B 0,C 180,E1 -16896.058,E2 -16896.058} C_VEL
LIN {X 0,Y 285.647,Z 153.993,A -85,B 0,C 180,E1 -16896.817,E2 -16896.817} C_VEL
LIN {X 0,Y 284.51,Z 151.609,A -85,B 0,C 180,E1 -16897.247,E2 -16897.247} C_VEL
LIN {X 0,Y 284.355,Z 150.869,A -85,B 0,C 180,E1 -16897.378,E2 -16897.378} C_VEL
LIN {X 0,Y 284.384,Z 150.685,A -85,B 0,C 180,E1 -16901.26,E2 -16901.26} C_VEL
LIN {X 0,Y 284.468,Z 150.67,A -85,B 0,C 180,E1 -16905.696,E2 -16905.696} C_VEL
LIN {X 0,Y 284.567,Z 150.662,A -85,B 0,C 180,E1 -16910.044,E2 -16910.044} C_VEL
LIN {X 0,Y 284.698,Z 150.648,A -85,B 0,C 180,E1 -16912.909,E2 -16912.909} C_VEL
LIN {X 0,Y 284.854,Z 150.619,A -85,B 0,C 180,E1 -16918.586,E2 -16918.586} C_VEL
LIN {X 0,Y 284.854,Z 150.618,A -85,B 0,C 180,E1 -16921.413,E2 -16921.413} C_VEL
LIN {X 0,Y 284.578,Z 150.653,A -85,B 0,C 180,E1 -16925.669,E2 -16925.669} C_VEL
LIN {X 0,Y 284.608,Z 150.648,A -85,B 0,C 180,E1 -16928.981,E2 -16928.981} C_VEL
LIN {X 0,Y 284.474,Z 150.665,A -85,B 0,C 180,E1 -16932.846,E2 -16932.846} C_VEL
LIN {X 0,Y 284.486,Z 150.663,A -85,B 0,C 180,E1 -16935.768,E2 -16935.768} C_VEL
LIN {X 0,Y 284.377,Z 150.679,A -85,B 0,C 180,E1 -16940.242,E2 -16940.242} C_VEL
LIN {X 0,Y 284.368,Z 150.683,A -85,B 0,C 180,E1 -16943.875,E2 -16943.875} C_VEL
LIN {X 0,Y 284.395,Z 150.681,A -85,B 0,C 180,E1 -16947.173,E2 -16947.173} C_VEL
LIN {X 0,Y 284.294,Z 150.695,A -85,B 0,C 180,E1 -16951.274,E2 -16951.274} C_VEL
LIN {X 0,Y 284.339,Z 150.687,A -85,B 0,C 180,E1 -16955.348,E2 -16955.348} C_VEL
LIN {X 0,Y 284.306,Z 150.767,A -85,B 0,C 180,E1 -16957.954,E2 -16957.954} C_VEL
LIN {X 0,Y 286.726,Z 157.451,A -85,B 0,C 180,E1 -16961.437,E2 -16961.437} C_VEL
LIN {X 0,Y 287.656,Z 160.21,A -85,B 0,C 180,E1 -16962.668,E2 -16962.668} C_VEL
LIN {X 0,Y 290.901,Z 165.014,A -85,B 0,C 180,E1 -16963.732,E2 -16963.732} C_VEL
LIN {X 0,Y 292.599,Z 167.471,A -85,B 0,C 180,E1 -16964.268,E2 -16964.268} C_VEL
LIN {X 0,Y 296.401,Z 173.237,A -85,B 0,C 180,E1 -16965.427,E2 -16965.427} C_VEL
LIN {X 0,Y 300.208,Z 179.149,A -85,B 0,C 180,E1 -16966.528,E2 -16966.528} C_VEL
LIN {X 0,Y 307.648,Z 191.568,A -85,B 0,C 180,E1 -16968.557,E2 -16968.557} C_VEL
LIN {X 0,Y 314.863,Z 205.433,A -85,B 0,C 180,E1 -16970.415,E2 -16970.415} C_VEL
LIN {X 0,Y 321.077,Z 218.943,A -85,B 0,C 180,E1 -16971.94,E2 -16971.94} C_VEL
LIN {X 0,Y 321.401,Z 221.193,A -85,B 0,C 180,E1 -16972.065,E2 -16972.065} C_VEL
LIN {X 0,Y 316.27,Z 328.444,A -85,B 0,C 180,E1 -16974.561,E2 -16974.561} C_VEL
LIN {X 0,Y 314.707,Z 343.211,A -85,B 0,C 180,E1 -16975.093,E2 -16975.093} C_VEL
LIN {X 0,Y 312.452,Z 358.382,A -85,B 0,C 180,E1 -16975.881,E2 -16975.881} C_VEL
LIN {X 0,Y 310.025,Z 371.973,A -85,B 0,C 180,E1 -16976.846,E2 -16976.846} C_VEL
LIN {X 0,Y 307.13,Z 385.256,A -85,B 0,C 180,E1 -16978.034,E2 -16978.034} C_VEL
LIN {X 0,Y 304.128,Z 397.783,A -85,B 0,C 180,E1 -16979.444,E2 -16979.444} C_VEL
LIN {X 0,Y 300.602,Z 410.418,A -85,B 0,C 180,E1 -16981.171,E2 -16981.171} C_VEL
LIN {X 0,Y 297.514,Z 421.039,A -85,B 0,C 180,E1 -16982.953,E2 -16982.953} C_VEL
LIN {X 0,Y 294.371,Z 430.954,A -85,B 0,C 180,E1 -16984.935,E2 -16984.935} C_VEL
LIN {X 0,Y 291.777,Z 439.355,A -85,B 0,C 180,E1 -16986.958,E2 -16986.958} C_VEL
LIN {X 0,Y 289.037,Z 447.657,A -85,B 0,C 180,E1 -16989.356,E2 -16989.356} C_VEL
LIN {X 0,Y 286.576,Z 455.492,A -85,B 0,C 180,E1 -16992.149,E2 -16992.149} C_VEL
LIN {X 0,Y 285.011,Z 460.348,A -85,B 0,C 180,E1 -16994.262,E2 -16994.262} C_VEL
LIN {X 0,Y 283.735,Z 465.611,A -85,B 0,C 180,E1 -16997.12,E2 -16997.12} C_VEL
LIN {X 0,Y 282.832,Z 469.579,A -85,B 0,C 180,E1 -16999.984,E2 -16999.984} C_VEL
LIN {X 0,Y 282.388,Z 472.315,A -85,B 0,C 180,E1 -17002.852,E2 -17002.852} C_VEL
LIN {X 0,Y 282.281,Z 473.903,A -85,B 0,C 180,E1 -17005.717,E2 -17005.717} C_VEL
LIN {X 0,Y 282.331,Z 474.365,A -85,B 0,C 180,E1 -17008.574,E2 -17008.574} C_VEL
LIN {X 0,Y 282.335,Z 473.684,A -85,B 0,C 180,E1 -17011.427,E2 -17011.427} C_VEL
LIN {X 0,Y 282.31,Z 471.78,A -85,B 0,C 180,E1 -17014.284,E2 -17014.284} C_VEL
LIN {X 0,Y 282.467,Z 468.651,A -85,B 0,C 180,E1 -17017.147,E2 -17017.147} C_VEL
LIN {X 0,Y 282.729,Z 464.22,A -85,B 0,C 180,E1 -17020.021,E2 -17020.021} C_VEL
LIN {X 0,Y 283.504,Z 458.384,A -85,B 0,C 180,E1 -17022.892,E2 -17022.892} C_VEL
LIN {X 0,Y 284.603,Z 450.963,A -85,B 0,C 180,E1 -17025.762,E2 -17025.762} C_VEL
LIN {X 0,Y 286.078,Z 443.001,A -85,B 0,C 180,E1 -17028.254,E2 -17028.254} C_VEL
LIN {X 0,Y 288.111,Z 433.419,A -85,B 0,C 180,E1 -17030.715,E2 -17030.715} C_VEL
LIN {X 0,Y 290.259,Z 422.314,A -85,B 0,C 180,E1 -17033.062,E2 -17033.062} C_VEL
LIN {X 0,Y 292.638,Z 410.865,A -85,B 0,C 180,E1 -17035.043,E2 -17035.043} C_VEL
LIN {X 0,Y 295.035,Z 397.747,A -85,B 0,C 180,E1 -17036.911,E2 -17036.911} C_VEL
LIN {X 0,Y 297.463,Z 384.764,A -85,B 0,C 180,E1 -17038.391,E2 -17038.391} C_VEL
LIN {X 0,Y 299.44,Z 371.614,A -85,B 0,C 180,E1 -17039.617,E2 -17039.617} C_VEL
LIN {X 0,Y 301.276,Z 357.114,A -85,B 0,C 180,E1 -17040.676,E2 -17040.676} C_VEL
LIN {X 0,Y 302.901,Z 342.259,A -85,B 0,C 180,E1 -17041.471,E2 -17041.471} C_VEL
LIN {X 0,Y 303.991,Z 327.309,A -85,B 0,C 180,E1 -17042.026,E2 -17042.026} C_VEL
LIN {X 0,Y 307.926,Z 217.259,A -85,B 0,C 180,E1 -17044.607,E2 -17044.607} C_VEL
LIN {X 0,Y 305.579,Z 203.344,A -85,B 0,C 180,E1 -17045.232,E2 -17045.232} C_VEL
LIN {X 0,Y 296.969,Z 182.562,A -85,B 0,C 180,E1 -17046.781,E2 -17046.781} C_VEL
LIN {X 0,Y 288.85,Z 165.094,A -85,B 0,C 180,E1 -17048.275,E2 -17048.275} C_VEL
LIN {X 0,Y 287.351,Z 161.731,A -85,B 0,C 180,E1 -17048.613,E2 -17048.613} C_VEL
LIN {X 0,Y 284.282,Z 150.701,A -85,B 0,C 180,E1 -17052.094,E2 -17052.094} C_VEL
LIN {X 0,Y 284.257,Z 150.706,A -85,B 0,C 180,E1 -17056.19,E2 -17056.19} C_VEL
LIN {X 0,Y 284.308,Z 150.689,A -85,B 0,C 180,E1 -17060.025,E2 -17060.025} C_VEL
LIN {X 0,Y 284.333,Z 150.692,A -85,B 0,C 180,E1 -17063.615,E2 -17063.615} C_VEL
LIN {X 0,Y 284.308,Z 150.692,A -85,B 0,C 180,E1 -17067.191,E2 -17067.191} C_VEL
LIN {X 0,Y 284.339,Z 150.681,A -85,B 0,C 180,E1 -17070.374,E2 -17070.374} C_VEL
LIN {X 0,Y 284.308,Z 150.672,A -85,B 0,C 180,E1 -17073.58,E2 -17073.58} C_VEL
LIN {X 0,Y 284.332,Z 150.692,A -85,B 0,C 180,E1 -17076.705,E2 -17076.705} C_VEL
LIN {X 0,Y 284.38,Z 150.683,A -85,B 0,C 180,E1 -17079.905,E2 -17079.905} C_VEL
LIN {X 0,Y 284.451,Z 150.674,A -85,B 0,C 180,E1 -17084.493,E2 -17084.493} C_VEL
LIN {X 0,Y 284.486,Z 150.668,A -85,B 0,C 180,E1 -17088.602,E2 -17088.602} C_VEL
LIN {X 0,Y 284.613,Z 150.653,A -85,B 0,C 180,E1 -17091.48,E2 -17091.48} C_VEL
LIN {X 0,Y 284.572,Z 150.663,A -85,B 0,C 180,E1 -17094.331,E2 -17094.331} C_VEL
LIN {X 0,Y 284.842,Z 150.595,A -85,B 0,C 180,E1 -17098.587,E2 -17098.587} C_VEL
LIN {X 0,Y 284.84,Z 150.608,A -85,B 0,C 180,E1 -17101.414,E2 -17101.414} C_VEL
LIN {X 0,Y 284.646,Z 150.637,A -85,B 0,C 180,E1 -17107.092,E2 -17107.092} C_VEL
LIN {X 0,Y 284.516,Z 150.63,A -85,B 0,C 180,E1 -17109.958,E2 -17109.958} C_VEL
LIN {X 0,Y 284.41,Z 150.681,A -85,B 0,C 180,E1 -17114.307,E2 -17114.307} C_VEL
LIN {X 0,Y 284.331,Z 150.683,A -85,B 0,C 180,E1 -17117.255,E2 -17117.255} C_VEL
LIN {X 0,Y 284.314,Z 150.692,A -85,B 0,C 180,E1 -17120.248,E2 -17120.248} C_VEL
LIN {X 0,Y 284.297,Z 150.698,A -85,B 0,C 180,E1 -17123.84,E2 -17123.84} C_VEL
LIN {X 0,Y 284.29,Z 150.681,A -85,B 0,C 180,E1 -17127.129,E2 -17127.129} C_VEL
LIN {X 0,Y 284.277,Z 150.665,A -85,B 0,C 180,E1 -17130.084,E2 -17130.084} C_VEL
LIN {X 0,Y 284.309,Z 150.69,A -85,B 0,C 180,E1 -17132.946,E2 -17132.946} C_VEL
LIN {X 0,Y 284.323,Z 150.677,A -85,B 0,C 180,E1 -17136.388,E2 -17136.388} C_VEL
LIN {X 0,Y 284.287,Z 150.682,A -85,B 0,C 180,E1 -17139.999,E2 -17139.999} C_VEL
LIN {X 0,Y 284.239,Z 150.692,A -85,B 0,C 180,E1 -17144.188,E2 -17144.188} C_VEL
LIN {X 0,Y 284.245,Z 150.698,A -85,B 0,C 180,E1 -17148.119,E2 -17148.119} C_VEL
LIN {X 0,Y 284.286,Z 150.681,A -85,B 0,C 180,E1 -17152.289,E2 -17152.289} C_VEL
LIN {X 0,Y 284.312,Z 150.694,A -85,B 0,C 180,E1 -17155.35,E2 -17155.35} C_VEL
LIN {X 0,Y 284.29,Z 150.693,A -85,B 0,C 180,E1 -17158.724,E2 -17158.724} C_VEL
LIN {X 0,Y 284.287,Z 150.691,A -85,B 0,C 180,E1 -17161.984,E2 -17161.984} C_VEL
LIN {X 0,Y 284.315,Z 150.697,A -85,B 0,C 180,E1 -17166.151,E2 -17166.151} C_VEL
LIN {X 0,Y 284.386,Z 150.686,A -85,B 0,C 180,E1 -17170.161,E2 -17170.161} C_VEL
LIN {X 0,Y 285.491,Z 153.625,A -85,B 0,C 180,E1 -17170.414,E2 -17170.414} C_VEL
LIN {X 0,Y 287.097,Z 156.324,A -85,B 0,C 180,E1 -17170.706,E2 -17170.706} C_VEL
LIN {X 0,Y 293.933,Z 168.578,A -85,B 0,C 180,E1 -17171.926,E2 -17171.926} C_VEL
LIN {X 0,Y 301.484,Z 184.979,A -85,B 0,C 180,E1 -17173.277,E2 -17173.277} C_VEL
LIN {X 0,Y 308.391,Z 201.755,A -85,B 0,C 180,E1 -17174.494,E2 -17174.494} C_VEL
LIN {X 0,Y 304.272,Z 313.556,A -85,B 0,C 180,E1 -17177.112,E2 -17177.112} C_VEL
LIN {X 0,Y 303.123,Z 329.481,A -85,B 0,C 180,E1 -17177.743,E2 -17177.743} C_VEL
LIN {X 0,Y 301.734,Z 343.944,A -85,B 0,C 180,E1 -17178.577,E2 -17178.577} C_VEL
LIN {X 0,Y 299.835,Z 358.717,A -85,B 0,C 180,E1 -17179.703,E2 -17179.703} C_VEL
LIN {X 0,Y 297.83,Z 372.075,A -85,B 0,C 180,E1 -17181.005,E2 -17181.005} C_VEL
LIN {X 0,Y 295.428,Z 385.722,A -85,B 0,C 180,E1 -17182.653,E2 -17182.653} C_VEL
LIN {X 0,Y 293.067,Z 398.067,A -85,B 0,C 180,E1 -17184.495,E2 -17184.495} C_VEL
LIN {X 0,Y 290.858,Z 409.294,A -85,B 0,C 180,E1 -17186.536,E2 -17186.536} C_VEL
LIN {X 0,Y 288.694,Z 419.886,A -85,B 0,C 180,E1 -17188.869,E2 -17188.869} C_VEL
LIN {X 0,Y 286.665,Z 429.335,A -85,B 0,C 180,E1 -17191.404,E2 -17191.404} C_VEL
LIN {X 0,Y 285.162,Z 436.881,A -85,B 0,C 180,E1 -17193.886,E2 -17193.886} C_VEL
LIN {X 0,Y 284.074,Z 443.113,A -85,B 0,C 180,E1 -17196.391,E2 -17196.391} C_VEL
LIN {X 0,Y 283.138,Z 448.85,A -85,B 0,C 180,E1 -17199.284,E2 -17199.284} C_VEL
LIN {X 0,Y 282.653,Z 452.278,A -85,B 0,C 180,E1 -17201.473,E2 -17201.473} C_VEL
LIN {X 0,Y 282.222,Z 455.652,A -85,B 0,C 180,E1 -17204.419,E2 -17204.419} C_VEL
LIN {X 0,Y 282.08,Z 457.76,A -85,B 0,C 180,E1 -17207.396,E2 -17207.396} C_VEL
LIN {X 0,Y 282.057,Z 458.634,A -85,B 0,C 180,E1 -17210.416,E2 -17210.416} C_VEL
LIN {X 0,Y 282.292,Z 458.241,A -85,B 0,C 180,E1 -17213.474,E2 -17213.474} C_VEL
LIN {X 0,Y 282.836,Z 456.537,A -85,B 0,C 180,E1 -17216.568,E2 -17216.568} C_VEL
LIN {X 0,Y 283.755,Z 453.443,A -85,B 0,C 180,E1 -17219.693,E2 -17219.693} C_VEL
LIN {X 0,Y 285.198,Z 448.855,A -85,B 0,C 180,E1 -17222.829,E2 -17222.829} C_VEL
LIN {X 0,Y 287.292,Z 442.633,A -85,B 0,C 180,E1 -17225.952,E2 -17225.952} C_VEL
LIN {X 0,Y 289.637,Z 435.658,A -85,B 0,C 180,E1 -17228.668,E2 -17228.668} C_VEL
LIN {X 0,Y 292.532,Z 427.04,A -85,B 0,C 180,E1 -17231.351,E2 -17231.351} C_VEL
LIN {X 0,Y 295.474,Z 418.098,A -85,B 0,C 180,E1 -17233.612,E2 -17233.612} C_VEL
LIN {X 0,Y 298.838,Z 407.398,A -85,B 0,C 180,E1 -17235.831,E2 -17235.831} C_VEL
LIN {X 0,Y 302.312,Z 395.521,A -85,B 0,C 180,E1 -17237.838,E2 -17237.838} C_VEL
LIN {X 0,Y 305.372,Z 384.111,A -85,B 0,C 180,E1 -17239.418,E2 -17239.418} C_VEL
LIN {X 0,Y 308.314,Z 371.915,A -85,B 0,C 180,E1 -17240.807,E2 -17240.807} C_VEL
LIN {X 0,Y 310.935,Z 358.893,A -85,B 0,C 180,E1 -17242.024,E2 -17242.024} C_VEL
LIN {X 0,Y 313.396,Z 344.53,A -85,B 0,C 180,E1 -17243.065,E2 -17243.065} C_VEL
LIN {X 0,Y 315.219,Z 330.792,A -85,B 0,C 180,E1 -17243.82,E2 -17243.82} C_VEL
LIN {X 0,Y 316.74,Z 315.118,A -85,B 0,C 180,E1 -17244.424,E2 -17244.424} C_VEL
LIN {X 0,Y 318.921,Z 270.746,A -85,B 0,C 180,E1 -17245.478,E2 -17245.478} C_VEL
LIN {X 0,Y 318.763,Z 264.949,A -85,B 0,C 180,E1 -17245.682,E2 -17245.682} C_VEL
LIN {X 0,Y 315.404,Z 246.416,A -85,B 0,C 180,E1 -17246.828,E2 -17246.828} C_VEL
LIN {X 0,Y 315.242,Z 240.62,A -85,B 0,C 180,E1 -17247.041,E2 -17247.041} C_VEL
LIN {X 0,Y 316.583,Z 214.006,A -85,B 0,C 180,E1 -17247.656,E2 -17247.656} C_VEL
LIN {X 0,Y 309.183,Z 199.244,A -85,B 0,C 180,E1 -17249.528,E2 -17249.528} C_VEL
LIN {X 0,Y 301.729,Z 186.289,A -85,B 0,C 180,E1 -17251.534,E2 -17251.534} C_VEL
LIN {X 0,Y 294.158,Z 174.587,A -85,B 0,C 180,E1 -17253.72,E2 -17253.72} C_VEL
LIN {X 0,Y 288.381,Z 166.556,A -85,B 0,C 180,E1 -17255.524,E2 -17255.524} C_VEL
LIN {X 0,Y 285.681,Z 163.111,A -85,B 0,C 180,E1 -17256.408,E2 -17256.408} C_VEL
LIN {X 0,Y 284.881,Z 161.97,A -85,B 0,C 180,E1 -17256.682,E2 -17256.682} C_VEL
LIN {X 0,Y 282.439,Z 159.334,A -85,B 0,C 180,E1 -17257.506,E2 -17257.506} C_VEL
LIN {X 0,Y 281.203,Z 157.074,A -85,B 0,C 180,E1 -17257.982,E2 -17257.982} C_VEL
LIN {X 0,Y 278.911,Z 155.277,A -85,B 0,C 180,E1 -17258.779,E2 -17258.779} C_VEL
LIN {X 0,Y 277.582,Z 152.875,A -85,B 0,C 180,E1 -17259.323,E2 -17259.323} C_VEL
LIN {X 0,Y 277.313,Z 151.561,A -85,B 0,C 180,E1 -17259.501,E2 -17259.501} C_VEL
LIN {X 0,Y 277.364,Z 151.561,A -85,B 0,C 180,E1 -17263.815,E2 -17263.815} C_VEL
LIN {X 0,Y 277.412,Z 151.555,A -85,B 0,C 180,E1 -17266.82,E2 -17266.82} C_VEL
LIN {X 0,Y 277.616,Z 151.52,A -85,B 0,C 180,E1 -17271.263,E2 -17271.263} C_VEL
LIN {X 0,Y 277.571,Z 151.525,A -85,B 0,C 180,E1 -17274.187,E2 -17274.187} C_VEL
LIN {X 0,Y 277.82,Z 151.495,A -85,B 0,C 180,E1 -17278.55,E2 -17278.55} C_VEL
LIN {X 0,Y 277.82,Z 151.494,A -85,B 0,C 180,E1 -17281.449,E2 -17281.449} C_VEL
LIN {X 0,Y 277.603,Z 151.532,A -85,B 0,C 180,E1 -17287.272,E2 -17287.272} C_VEL
LIN {X 0,Y 277.456,Z 151.547,A -85,B 0,C 180,E1 -17290.213,E2 -17290.213} C_VEL
LIN {X 0,Y 277.433,Z 151.552,A -85,B 0,C 180,E1 -17294.674,E2 -17294.674} C_VEL
LIN {X 0,Y 277.344,Z 151.553,A -85,B 0,C 180,E1 -17299.233,E2 -17299.233} C_VEL
LIN {X 0,Y 277.318,Z 151.564,A -85,B 0,C 180,E1 -17304.17,E2 -17304.17} C_VEL
LIN {X 0,Y 277.324,Z 151.565,A -85,B 0,C 180,E1 -17307.505,E2 -17307.505} C_VEL
LIN {X 0,Y 277.27,Z 151.571,A -85,B 0,C 180,E1 -17310.481,E2 -17310.481} C_VEL
LIN {X 0,Y 277.245,Z 151.575,A -85,B 0,C 180,E1 -17313.895,E2 -17313.895} C_VEL
LIN {X 0,Y 277.335,Z 151.78,A -85,B 0,C 180,E1 -17316.111,E2 -17316.111} C_VEL
LIN {X 0,Y 279.7,Z 158.441,A -85,B 0,C 180,E1 -17319.846,E2 -17319.846} C_VEL
LIN {X 0,Y 280.293,Z 159.977,A -85,B 0,C 180,E1 -17320.536,E2 -17320.536} C_VEL
LIN {X 0,Y 285.314,Z 167.164,A -85,B 0,C 180,E1 -17322.324,E2 -17322.324} C_VEL
LIN {X 0,Y 289.17,Z 172.683,A -85,B 0,C 180,E1 -17323.6,E2 -17323.6} C_VEL
LIN {X 0,Y 293.334,Z 179.178,A -85,B 0,C 180,E1 -17324.921,E2 -17324.921} C_VEL
LIN {X 0,Y 298.601,Z 187.541,A -85,B 0,C 180,E1 -17326.478,E2 -17326.478} C_VEL
LIN {X 0,Y 305.435,Z 199.627,A -85,B 0,C 180,E1 -17328.389,E2 -17328.389} C_VEL
LIN {X 0,Y 311.798,Z 212.378,A -85,B 0,C 180,E1 -17330.074,E2 -17330.074} C_VEL
LIN {X 0,Y 316.198,Z 222.198,A -85,B 0,C 180,E1 -17331.197,E2 -17331.197} C_VEL
LIN {X 0,Y 311.018,Z 327.063,A -85,B 0,C 180,E1 -17333.669,E2 -17333.669} C_VEL
LIN {X 0,Y 309.317,Z 343.058,A -85,B 0,C 180,E1 -17334.243,E2 -17334.243} C_VEL
LIN {X 0,Y 306.884,Z 358.787,A -85,B 0,C 180,E1 -17335.074,E2 -17335.074} C_VEL
LIN {X 0,Y 304.195,Z 373.216,A -85,B 0,C 180,E1 -17336.126,E2 -17336.126} C_VEL
LIN {X 0,Y 300.795,Z 387.838,A -85,B 0,C 180,E1 -17337.494,E2 -17337.494} C_VEL
LIN {X 0,Y 297.426,Z 401.02,A -85,B 0,C 180,E1 -17339.074,E2 -17339.074} C_VEL
LIN {X 0,Y 294.132,Z 412.085,A -85,B 0,C 180,E1 -17340.671,E2 -17340.671} C_VEL
LIN {X 0,Y 290.656,Z 423.276,A -85,B 0,C 180,E1 -17342.651,E2 -17342.651} C_VEL
LIN {X 0,Y 287.435,Z 432.748,A -85,B 0,C 180,E1 -17344.668,E2 -17344.668} C_VEL
LIN {X 0,Y 284.379,Z 442.089,A -85,B 0,C 180,E1 -17347.093,E2 -17347.093} C_VEL
LIN {X 0,Y 281.651,Z 449.93,A -85,B 0,C 180,E1 -17349.554,E2 -17349.554} C_VEL
LIN {X 0,Y 279.194,Z 457.287,A -85,B 0,C 180,E1 -17352.419,E2 -17352.419} C_VEL
LIN {X 0,Y 277.365,Z 463.165,A -85,B 0,C 180,E1 -17355.323,E2 -17355.323} C_VEL
LIN {X 0,Y 276.17,Z 467.721,A -85,B 0,C 180,E1 -17358.254,E2 -17358.254} C_VEL
LIN {X 0,Y 275.498,Z 471.017,A -85,B 0,C 180,E1 -17361.196,E2 -17361.196} C_VEL
LIN {X 0,Y 275.234,Z 473.454,A -85,B 0,C 180,E1 -17364.774,E2 -17364.774} C_VEL
LIN {X 0,Y 275.229,Z 474.089,A -85,B 0,C 180,E1 -17367.073,E2 -17367.073} C_VEL
LIN {X 0,Y 275.276,Z 473.93,A -85,B 0,C 180,E1 -17370.001,E2 -17370.001} C_VEL
LIN {X 0,Y 275.259,Z 472.612,A -85,B 0,C 180,E1 -17372.928,E2 -17372.928} C_VEL
LIN {X 0,Y 275.292,Z 470.049,A -85,B 0,C 180,E1 -17375.862,E2 -17375.862} C_VEL
LIN {X 0,Y 275.489,Z 466.223,A -85,B 0,C 180,E1 -17378.805,E2 -17378.805} C_VEL
LIN {X 0,Y 275.998,Z 461.042,A -85,B 0,C 180,E1 -17381.755,E2 -17381.755} C_VEL
LIN {X 0,Y 277.058,Z 454.374,A -85,B 0,C 180,E1 -17384.695,E2 -17384.695} C_VEL
LIN {X 0,Y 278.337,Z 447.156,A -85,B 0,C 180,E1 -17387.259,E2 -17387.259} C_VEL
LIN {X 0,Y 280.062,Z 438.447,A -85,B 0,C 180,E1 -17389.803,E2 -17389.803} C_VEL
LIN {X 0,Y 281.999,Z 429.602,A -85,B 0,C 180,E1 -17391.953,E2 -17391.953} C_VEL
LIN {X 0,Y 284.3,Z 418.433,A -85,B 0,C 180,E1 -17394.209,E2 -17394.209} C_VEL
LIN {X 0,Y 286.76,Z 406.555,A -85,B 0,C 180,E1 -17396.178,E2 -17396.178} C_VEL
LIN {X 0,Y 289.155,Z 393.931,A -85,B 0,C 180,E1 -17397.897,E2 -17397.897} C_VEL
LIN {X 0,Y 291.669,Z 380.107,A -85,B 0,C 180,E1 -17399.404,E2 -17399.404} C_VEL
LIN {X 0,Y 293.873,Z 365.268,A -85,B 0,C 180,E1 -17400.684,E2 -17400.684} C_VEL
LIN {X 0,Y 295.647,Z 350.868,A -85,B 0,C 180,E1 -17401.633,E2 -17401.633} C_VEL
LIN {X 0,Y 297.106,Z 335.525,A -85,B 0,C 180,E1 -17402.358,E2 -17402.358} C_VEL
LIN {X 0,Y 298.034,Z 319.459,A -85,B 0,C 180,E1 -17402.846,E2 -17402.846} C_VEL
LIN {X 0,Y 301.714,Z 218.262,A -85,B 0,C 180,E1 -17405.242,E2 -17405.242} C_VEL
LIN {X 0,Y 299.568,Z 205.631,A -85,B 0,C 180,E1 -17405.831,E2 -17405.831} C_VEL
LIN {X 0,Y 290.785,Z 184.434,A -85,B 0,C 180,E1 -17407.466,E2 -17407.466} C_VEL
LIN {X 0,Y 281.874,Z 165.421,A -85,B 0,C 180,E1 -17409.172,E2 -17409.172} C_VEL
LIN {X 0,Y 280.032,Z 161.602,A -85,B 0,C 180,E1 -17409.561,E2 -17409.561} C_VEL
LIN {X 0,Y 277.205,Z 151.582,A -85,B 0,C 180,E1 -17412.877,E2 -17412.877} C_VEL
LIN {X 0,Y 277.216,Z 151.583,A -85,B 0,C 180,E1 -17417.326,E2 -17417.326} C_VEL
LIN {X 0,Y 277.264,Z 151.564,A -85,B 0,C 180,E1 -17421.794,E2 -17421.794} C_VEL
LIN {X 0,Y 277.286,Z 151.566,A -85,B 0,C 180,E1 -17424.342,E2 -17424.342} C_VEL
LIN {X 0,Y 277.242,Z 151.573,A -85,B 0,C 180,E1 -17427.837,E2 -17427.837} C_VEL
LIN {X 0,Y 277.242,Z 151.552,A -85,B 0,C 180,E1 -17431.208,E2 -17431.208} C_VEL
LIN {X 0,Y 277.249,Z 151.563,A -85,B 0,C 180,E1 -17434.474,E2 -17434.474} C_VEL
LIN {X 0,Y 277.267,Z 151.564,A -85,B 0,C 180,E1 -17437.654,E2 -17437.654} C_VEL
LIN {X 0,Y 277.328,Z 151.566,A -85,B 0,C 180,E1 -17440.766,E2 -17440.766} C_VEL
LIN {X 0,Y 277.413,Z 151.554,A -85,B 0,C 180,E1 -17445.325,E2 -17445.325} C_VEL
LIN {X 0,Y 277.461,Z 151.547,A -85,B 0,C 180,E1 -17449.788,E2 -17449.788} C_VEL
LIN {X 0,Y 277.605,Z 151.524,A -85,B 0,C 180,E1 -17452.728,E2 -17452.728} C_VEL
LIN {X 0,Y 277.809,Z 151.471,A -85,B 0,C 180,E1 -17458.551,E2 -17458.551} C_VEL
LIN {X 0,Y 277.807,Z 151.484,A -85,B 0,C 180,E1 -17461.45,E2 -17461.45} C_VEL
LIN {X 0,Y 277.605,Z 151.51,A -85,B 0,C 180,E1 -17467.273,E2 -17467.273} C_VEL
LIN {X 0,Y 277.456,Z 151.51,A -85,B 0,C 180,E1 -17470.214,E2 -17470.214} C_VEL
LIN {X 0,Y 277.369,Z 151.557,A -85,B 0,C 180,E1 -17474.678,E2 -17474.678} C_VEL
LIN {X 0,Y 277.267,Z 151.571,A -85,B 0,C 180,E1 -17479.24,E2 -17479.24} C_VEL
LIN {X 0,Y 277.259,Z 151.574,A -85,B 0,C 180,E1 -17483.928,E2 -17483.928} C_VEL
LIN {X 0,Y 277.239,Z 151.556,A -85,B 0,C 180,E1 -17487.469,E2 -17487.469} C_VEL
LIN {X 0,Y 277.233,Z 151.545,A -85,B 0,C 180,E1 -17490.466,E2 -17490.466} C_VEL
LIN {X 0,Y 277.251,Z 151.573,A -85,B 0,C 180,E1 -17493.896,E2 -17493.896} C_VEL
LIN {X 0,Y 277.255,Z 151.544,A -85,B 0,C 180,E1 -17497.472,E2 -17497.472} C_VEL
LIN {X 0,Y 277.189,Z 151.578,A -85,B 0,C 180,E1 -17501.241,E2 -17501.241} C_VEL
LIN {X 0,Y 277.178,Z 151.559,A -85,B 0,C 180,E1 -17505.232,E2 -17505.232} C_VEL
LIN {X 0,Y 277.182,Z 151.583,A -85,B 0,C 180,E1 -17508.757,E2 -17508.757} C_VEL
LIN {X 0,Y 277.237,Z 151.559,A -85,B 0,C 180,E1 -17512.525,E2 -17512.525} C_VEL
LIN {X 0,Y 277.251,Z 151.569,A -85,B 0,C 180,E1 -17516.104,E2 -17516.104} C_VEL
LIN {X 0,Y 277.267,Z 151.575,A -85,B 0,C 180,E1 -17519.538,E2 -17519.538} C_VEL
LIN {X 0,Y 277.294,Z 151.569,A -85,B 0,C 180,E1 -17522.856,E2 -17522.856} C_VEL
LIN {X 0,Y 277.277,Z 151.574,A -85,B 0,C 180,E1 -17526.074,E2 -17526.074} C_VEL
LIN {X 0,Y 277.327,Z 151.711,A -85,B 0,C 180,E1 -17529.248,E2 -17529.248} C_VEL
LIN {X 0,Y 278.395,Z 154.56,A -85,B 0,C 180,E1 -17529.486,E2 -17529.486} C_VEL
LIN {X 0,Y 279.87,Z 156.757,A -85,B 0,C 180,E1 -17529.758,E2 -17529.758} C_VEL
LIN {X 0,Y 288.211,Z 171.524,A -85,B 0,C 180,E1 -17531.304,E2 -17531.304} C_VEL
LIN {X 0,Y 296.266,Z 189.167,A -85,B 0,C 180,E1 -17532.793,E2 -17532.793} C_VEL
LIN {X 0,Y 302.034,Z 203.147,A -85,B 0,C 180,E1 -17533.844,E2 -17533.844} C_VEL
LIN {X 0,Y 299.956,Z 261.839,A -85,B 0,C 180,E1 -17535.24,E2 -17535.24} C_VEL
LIN {X 0,Y 297.86,Z 314.675,A -85,B 0,C 180,E1 -17536.526,E2 -17536.526} C_VEL
LIN {X 0,Y 296.731,Z 330.221,A -85,B 0,C 180,E1 -17537.17,E2 -17537.17} C_VEL
LIN {X 0,Y 295.449,Z 343.075,A -85,B 0,C 180,E1 -17537.921,E2 -17537.921} C_VEL
LIN {X 0,Y 293.673,Z 356.829,A -85,B 0,C 180,E1 -17538.962,E2 -17538.962} C_VEL
LIN {X 0,Y 291.601,Z 370.574,A -85,B 0,C 180,E1 -17540.287,E2 -17540.287} C_VEL
LIN {X 0,Y 289.351,Z 383.24,A -85,B 0,C 180,E1 -17541.795,E2 -17541.795} C_VEL
LIN {X 0,Y 287.071,Z 394.979,A -85,B 0,C 180,E1 -17543.498,E2 -17543.498} C_VEL
LIN {X 0,Y 284.827,Z 405.874,A -85,B 0,C 180,E1 -17545.4,E2 -17545.4} C_VEL
LIN {X 0,Y 282.625,Z 415.96,A -85,B 0,C 180,E1 -17547.505,E2 -17547.505} C_VEL
LIN {X 0,Y 281.014,Z 423.859,A -85,B 0,C 180,E1 -17549.475,E2 -17549.475} C_VEL
LIN {X 0,Y 279.267,Z 431.775,A -85,B 0,C 180,E1 -17551.802,E2 -17551.802} C_VEL
LIN {X 0,Y 277.82,Z 438.961,A -85,B 0,C 180,E1 -17554.352,E2 -17554.352} C_VEL
LIN {X 0,Y 276.625,Z 445.631,A -85,B 0,C 180,E1 -17557.298,E2 -17557.298} C_VEL
LIN {X 0,Y 275.812,Z 450.84,A -85,B 0,C 180,E1 -17560.274,E2 -17560.274} C_VEL
LIN {X 0,Y 275.285,Z 454.712,A -85,B 0,C 180,E1 -17563.283,E2 -17563.283} C_VEL
LIN {X 0,Y 274.996,Z 457.322,A -85,B 0,C 180,E1 -17566.327,E2 -17566.327} C_VEL
LIN {X 0,Y 274.967,Z 458.681,A -85,B 0,C 180,E1 -17569.406,E2 -17569.406} C_VEL
LIN {X 0,Y 275.125,Z 458.764,A -85,B 0,C 180,E1 -17572.53,E2 -17572.53} C_VEL
LIN {X 0,Y 275.559,Z 457.555,A -85,B 0,C 180,E1 -17575.694,E2 -17575.694} C_VEL
LIN {X 0,Y 276.377,Z 454.994,A -85,B 0,C 180,E1 -17578.891,E2 -17578.891} C_VEL
LIN {X 0,Y 277.716,Z 450.983,A -85,B 0,C 180,E1 -17582.102,E2 -17582.102} C_VEL
LIN {X 0,Y 279.688,Z 445.404,A -85,B 0,C 180,E1 -17585.306,E2 -17585.306} C_VEL
LIN {X 0,Y 281.573,Z 440.038,A -85,B 0,C 180,E1 -17587.699,E2 -17587.699} C_VEL
LIN {X 0,Y 284.319,Z 432.395,A -85,B 0,C 180,E1 -17590.456,E2 -17590.456} C_VEL
LIN {X 0,Y 287.611,Z 422.996,A -85,B 0,C 180,E1 -17593.172,E2 -17593.172} C_VEL
LIN {X 0,Y 291.181,Z 412.625,A -85,B 0,C 180,E1 -17595.576,E2 -17595.576} C_VEL
LIN {X 0,Y 294.678,Z 401.534,A -85,B 0,C 180,E1 -17597.675,E2 -17597.675} C_VEL
LIN {X 0,Y 298.123,Z 389.783,A -85,B 0,C 180,E1 -17599.487,E2 -17599.487} C_VEL
LIN {X 0,Y 301.54,Z 376.757,A -85,B 0,C 180,E1 -17601.119,E2 -17601.119} C_VEL
LIN {X 0,Y 304.525,Z 363.187,A -85,B 0,C 180,E1 -17602.497,E2 -17602.497} C_VEL
LIN {X 0,Y 307.21,Z 349.102,A -85,B 0,C 180,E1 -17603.607,E2 -17603.607} C_VEL
LIN {X 0,Y 309.382,Z 334.192,A -85,B 0,C 180,E1 -17604.511,E2 -17604.511} C_VEL
LIN {X 0,Y 311.166,Z 318.132,A -85,B 0,C 180,E1 -17605.18,E2 -17605.18} C_VEL
LIN {X 0,Y 312.326,Z 299.229,A -85,B 0,C 180,E1 -17605.683,E2 -17605.683} C_VEL
LIN {X 0,Y 315.242,Z 240.62,A -85,B 0,C 180,E1 -17607.041,E2 -17607.041} C_VEL
LIN {X 0,Y 315.256,Z 234.74,A -85,B 0,C 180,E1 -17607.227,E2 -17607.227} C_VEL
LIN {X 0,Y 314.647,Z 229.016,A -85,B 0,C 180,E1 -17607.519,E2 -17607.519} C_VEL
LIN {X 0,Y 313.023,Z 221.748,A -85,B 0,C 180,E1 -17608.05,E2 -17608.05} C_VEL
LIN {X 0,Y 310.62,Z 215.018,A -85,B 0,C 180,E1 -17608.719,E2 -17608.719} C_VEL
LIN {X 0,Y 309.167,Z 211.899,A -85,B 0,C 180,E1 -17609.101,E2 -17609.101} C_VEL
LIN {X 0,Y 303.284,Z 200.597,A -85,B 0,C 180,E1 -17610.683,E2 -17610.683} C_VEL
LIN {X 0,Y 297.069,Z 189.79,A -85,B 0,C 180,E1 -17612.449,E2 -17612.449} C_VEL
LIN {X 0,Y 289.498,Z 177.964,A -85,B 0,C 180,E1 -17614.754,E2 -17614.754} C_VEL
LIN {X 0,Y 285.238,Z 172.261,A -85,B 0,C 180,E1 -17616.134,E2 -17616.134} C_VEL
LIN {X 0,Y 281.937,Z 167.894,A -85,B 0,C 180,E1 -17617.267,E2 -17617.267} C_VEL
LIN {X 0,Y 279.3,Z 164.698,A -85,B 0,C 180,E1 -17618.212,E2 -17618.212} C_VEL
LIN {X 0,Y 278.413,Z 163.26,A -85,B 0,C 180,E1 -17618.556,E2 -17618.556} C_VEL
LIN {X 0,Y 275.849,Z 160.722,A -85,B 0,C 180,E1 -17619.506,E2 -17619.506} C_VEL
LIN {X 0,Y 274.34,Z 158.012,A -85,B 0,C 180,E1 -17620.149,E2 -17620.149} C_VEL
LIN {X 0,Y 271.89,Z 156.146,A -85,B 0,C 180,E1 -17621.099,E2 -17621.099} C_VEL
LIN {X 0,Y 270.594,Z 153.821,A -85,B 0,C 180,E1 -17621.693,E2 -17621.693} C_VEL
LIN {X 0,Y 270.282,Z 152.437,A -85,B 0,C 180,E1 -17621.916,E2 -17621.916} C_VEL
LIN {X 0,Y 270.373,Z 152.424,A -85,B 0,C 180,E1 -17624.933,E2 -17624.933} C_VEL
LIN {X 0,Y 270.442,Z 152.424,A -85,B 0,C 180,E1 -17629.518,E2 -17629.518} C_VEL
LIN {X 0,Y 270.611,Z 152.401,A -85,B 0,C 180,E1 -17632.538,E2 -17632.538} C_VEL
LIN {X 0,Y 270.786,Z 152.37,A -85,B 0,C 180,E1 -17638.512,E2 -17638.512} C_VEL
LIN {X 0,Y 270.786,Z 152.37,A -85,B 0,C 180,E1 -17641.487,E2 -17641.487} C_VEL
LIN {X 0,Y 270.564,Z 152.407,A -85,B 0,C 180,E1 -17647.462,E2 -17647.462} C_VEL
LIN {X 0,Y 270.409,Z 152.427,A -85,B 0,C 180,E1 -17650.482,E2 -17650.482} C_VEL
LIN {X 0,Y 270.402,Z 152.423,A -85,B 0,C 180,E1 -17655.064,E2 -17655.064} C_VEL
LIN {X 0,Y 270.3,Z 152.43,A -85,B 0,C 180,E1 -17659.755,E2 -17659.755} C_VEL
LIN {X 0,Y 270.272,Z 152.445,A -85,B 0,C 180,E1 -17664.585,E2 -17664.585} C_VEL
LIN {X 0,Y 270.268,Z 152.446,A -85,B 0,C 180,E1 -17667.908,E2 -17667.908} C_VEL
LIN {X 0,Y 270.182,Z 152.452,A -85,B 0,C 180,E1 -17671.348,E2 -17671.348} C_VEL
LIN {X 0,Y 270.224,Z 152.549,A -85,B 0,C 180,E1 -17673.869,E2 -17673.869} C_VEL
LIN {X 0,Y 271.831,Z 157.1,A -85,B 0,C 180,E1 -17676.729,E2 -17676.729} C_VEL
LIN {X 0,Y 272.836,Z 159.498,A -85,B 0,C 180,E1 -17678.068,E2 -17678.068} C_VEL
LIN {X 0,Y 276.006,Z 164.088,A -85,B 0,C 180,E1 -17679.371,E2 -17679.371} C_VEL
LIN {X 0,Y 278.056,Z 166.758,A -85,B 0,C 180,E1 -17680.159,E2 -17680.159} C_VEL
LIN {X 0,Y 282.288,Z 172.859,A -85,B 0,C 180,E1 -17681.72,E2 -17681.72} C_VEL
LIN {X 0,Y 286.233,Z 178.642,A -85,B 0,C 180,E1 -17683.07,E2 -17683.07} C_VEL
LIN {X 0,Y 292.579,Z 188.682,A -85,B 0,C 180,E1 -17685.11,E2 -17685.11} C_VEL
LIN {X 0,Y 299.909,Z 201.368,A -85,B 0,C 180,E1 -17687.28,E2 -17687.28} C_VEL
LIN {X 0,Y 306.525,Z 214.525,A -85,B 0,C 180,E1 -17689.13,E2 -17689.13} C_VEL
LIN {X 0,Y 311.099,Z 225.007,A -85,B 0,C 180,E1 -17690.362,E2 -17690.362} C_VEL
LIN {X 0,Y 305.756,Z 327.2,A -85,B 0,C 180,E1 -17692.785,E2 -17692.785} C_VEL
LIN {X 0,Y 304.006,Z 343.025,A -85,B 0,C 180,E1 -17693.364,E2 -17693.364} C_VEL
LIN {X 0,Y 301.62,Z 358.109,A -85,B 0,C 180,E1 -17694.167,E2 -17694.167} C_VEL
LIN {X 0,Y 298.781,Z 372.626,A -85,B 0,C 180,E1 -17695.221,E2 -17695.221} C_VEL
LIN {X 0,Y 295.304,Z 387.166,A -85,B 0,C 180,E1 -17696.588,E2 -17696.588} C_VEL
LIN {X 0,Y 291.78,Z 400.545,A -85,B 0,C 180,E1 -17698.205,E2 -17698.205} C_VEL
LIN {X 0,Y 288,Z 412.671,A -85,B 0,C 180,E1 -17699.984,E2 -17699.984} C_VEL
LIN {X 0,Y 284.372,Z 423.753,A -85,B 0,C 180,E1 -17701.994,E2 -17701.994} C_VEL
LIN {X 0,Y 280.287,Z 435.054,A -85,B 0,C 180,E1 -17704.511,E2 -17704.511} C_VEL
LIN {X 0,Y 277.372,Z 443.584,A -85,B 0,C 180,E1 -17706.876,E2 -17706.876} C_VEL
LIN {X 0,Y 274.263,Z 452.111,A -85,B 0,C 180,E1 -17709.761,E2 -17709.761} C_VEL
LIN {X 0,Y 271.816,Z 458.99,A -85,B 0,C 180,E1 -17712.703,E2 -17712.703} C_VEL
LIN {X 0,Y 270.13,Z 464.436,A -85,B 0,C 180,E1 -17715.691,E2 -17715.691} C_VEL
LIN {X 0,Y 269.168,Z 467.679,A -85,B 0,C 180,E1 -17717.944,E2 -17717.944} C_VEL
LIN {X 0,Y 268.44,Z 470.944,A -85,B 0,C 180,E1 -17720.963,E2 -17720.963} C_VEL
LIN {X 0,Y 268.143,Z 472.987,A -85,B 0,C 180,E1 -17723.983,E2 -17723.983} C_VEL
LIN {X 0,Y 268.14,Z 473.902,A -85,B 0,C 180,E1 -17726.996,E2 -17726.996} C_VEL
LIN {X 0,Y 268.199,Z 473.689,A -85,B 0,C 180,E1 -17730.001,E2 -17730.001} C_VEL
LIN {X 0,Y 268.169,Z 472.318,A -85,B 0,C 180,E1 -17733.005,E2 -17733.005} C_VEL
LIN {X 0,Y 268.213,Z 469.723,A -85,B 0,C 180,E1 -17736.017,E2 -17736.017} C_VEL
LIN {X 0,Y 268.422,Z 465.835,A -85,B 0,C 180,E1 -17739.039,E2 -17739.039} C_VEL
LIN {X 0,Y 268.997,Z 460.586,A -85,B 0,C 180,E1 -17742.065,E2 -17742.065} C_VEL
LIN {X 0,Y 270.079,Z 453.841,A -85,B 0,C 180,E1 -17745.084,E2 -17745.084} C_VEL
LIN {X 0,Y 271.481,Z 446.543,A -85,B 0,C 180,E1 -17747.71,E2 -17747.71} C_VEL
LIN {X 0,Y 273.32,Z 437.746,A -85,B 0,C 180,E1 -17750.313,E2 -17750.313} C_VEL
LIN {X 0,Y 275.662,Z 427.346,A -85,B 0,C 180,E1 -17752.831,E2 -17752.831} C_VEL
LIN {X 0,Y 278.033,Z 416.216,A -85,B 0,C 180,E1 -17755.05,E2 -17755.05} C_VEL
LIN {X 0,Y 280.563,Z 404.289,A -85,B 0,C 180,E1 -17757.003,E2 -17757.003} C_VEL
LIN {X 0,Y 282.84,Z 392.676,A -85,B 0,C 180,E1 -17758.577,E2 -17758.577} C_VEL
LIN {X 0,Y 285.372,Z 378.941,A -85,B 0,C 180,E1 -17760.08,E2 -17760.08} C_VEL
LIN {X 0,Y 287.562,Z 364.423,A -85,B 0,C 180,E1 -17761.34,E2 -17761.34} C_VEL
LIN {X 0,Y 289.21,Z 351.599,A -85,B 0,C 180,E1 -17762.205,E2 -17762.205} C_VEL
LIN {X 0,Y 290.735,Z 336.466,A -85,B 0,C 180,E1 -17762.95,E2 -17762.95} C_VEL
LIN {X 0,Y 291.692,Z 321.112,A -85,B 0,C 180,E1 -17763.447,E2 -17763.447} C_VEL
LIN {X 0,Y 295.544,Z 219.205,A -85,B 0,C 180,E1 -17765.905,E2 -17765.905} C_VEL
LIN {X 0,Y 293.747,Z 208.358,A -85,B 0,C 180,E1 -17766.422,E2 -17766.422} C_VEL
LIN {X 0,Y 285.294,Z 187.922,A -85,B 0,C 180,E1 -17768.046,E2 -17768.046} C_VEL
LIN {X 0,Y 276.85,Z 169.679,A -85,B 0,C 180,E1 -17769.725,E2 -17769.725} C_VEL
LIN {X 0,Y 272.708,Z 161.266,A -85,B 0,C 180,E1 -17770.63,E2 -17770.63} C_VEL
LIN {X 0,Y 270.155,Z 152.463,A -85,B 0,C 180,E1 -17773.625,E2 -17773.625} C_VEL
LIN {X 0,Y 270.173,Z 152.46,A -85,B 0,C 180,E1 -17777.443,E2 -17777.443} C_VEL
LIN {X 0,Y 270.209,Z 152.44,A -85,B 0,C 180,E1 -17781.375,E2 -17781.375} C_VEL
LIN {X 0,Y 270.204,Z 152.45,A -85,B 0,C 180,E1 -17785.095,E2 -17785.095} C_VEL
LIN {X 0,Y 270.186,Z 152.454,A -85,B 0,C 180,E1 -17789.137,E2 -17789.137} C_VEL
LIN {X 0,Y 270.225,Z 152.418,A -85,B 0,C 180,E1 -17792.164,E2 -17792.164} C_VEL
LIN {X 0,Y 270.23,Z 152.447,A -85,B 0,C 180,E1 -17795.543,E2 -17795.543} C_VEL
LIN {X 0,Y 270.265,Z 152.442,A -85,B 0,C 180,E1 -17800.242,E2 -17800.242} C_VEL
LIN {X 0,Y 270.381,Z 152.431,A -85,B 0,C 180,E1 -17804.935,E2 -17804.935} C_VEL
LIN {X 0,Y 270.414,Z 152.425,A -85,B 0,C 180,E1 -17809.518,E2 -17809.518} C_VEL
LIN {X 0,Y 270.566,Z 152.399,A -85,B 0,C 180,E1 -17812.538,E2 -17812.538} C_VEL
LIN {X 0,Y 270.774,Z 152.346,A -85,B 0,C 180,E1 -17818.513,E2 -17818.513} C_VEL
LIN {X 0,Y 270.772,Z 152.359,A -85,B 0,C 180,E1 -17821.488,E2 -17821.488} C_VEL
LIN {X 0,Y 270.567,Z 152.382,A -85,B 0,C 180,E1 -17827.463,E2 -17827.463} C_VEL
LIN {X 0,Y 270.387,Z 152.392,A -85,B 0,C 180,E1 -17830.484,E2 -17830.484} C_VEL
LIN {X 0,Y 270.34,Z 152.433,A -85,B 0,C 180,E1 -17835.069,E2 -17835.069} C_VEL
LIN {X 0,Y 270.212,Z 152.452,A -85,B 0,C 180,E1 -17839.763,E2 -17839.763} C_VEL
LIN {X 0,Y 270.186,Z 152.454,A -85,B 0,C 180,E1 -17844.436,E2 -17844.436} C_VEL
LIN {X 0,Y 270.189,Z 152.428,A -85,B 0,C 180,E1 -17847.919,E2 -17847.919} C_VEL
LIN {X 0,Y 270.173,Z 152.434,A -85,B 0,C 180,E1 -17851.35,E2 -17851.35} C_VEL
LIN {X 0,Y 270.202,Z 152.45,A -85,B 0,C 180,E1 -17854.906,E2 -17854.906} C_VEL
LIN {X 0,Y 270.203,Z 152.42,A -85,B 0,C 180,E1 -17858.71,E2 -17858.71} C_VEL
LIN {X 0,Y 270.153,Z 152.454,A -85,B 0,C 180,E1 -17863.245,E2 -17863.245} C_VEL
LIN {X 0,Y 270.156,Z 152.444,A -85,B 0,C 180,E1 -17867.438,E2 -17867.438} C_VEL
LIN {X 0,Y 270.156,Z 152.444,A -85,B 0,C 180,E1 -17871.365,E2 -17871.365} C_VEL
LIN {X 0,Y 270.203,Z 152.453,A -85,B 0,C 180,E1 -17875.094,E2 -17875.094} C_VEL
LIN {X 0,Y 270.189,Z 152.456,A -85,B 0,C 180,E1 -17879.136,E2 -17879.136} C_VEL
LIN {X 0,Y 270.227,Z 152.443,A -85,B 0,C 180,E1 -17882.163,E2 -17882.163} C_VEL
LIN {X 0,Y 270.222,Z 152.455,A -85,B 0,C 180,E1 -17885.547,E2 -17885.547} C_VEL
LIN {X 0,Y 270.211,Z 152.453,A -85,B 0,C 180,E1 -17888.237,E2 -17888.237} C_VEL
LIN {X 0,Y 271.16,Z 155.219,A -85,B 0,C 180,E1 -17888.47,E2 -17888.47} C_VEL
LIN {X 0,Y 272.685,Z 157.447,A -85,B 0,C 180,E1 -17888.766,E2 -17888.766} C_VEL
LIN {X 0,Y 282.185,Z 173.846,A -85,B 0,C 180,E1 -17890.594,E2 -17890.594} C_VEL
LIN {X 0,Y 289.734,Z 190.222,A -85,B 0,C 180,E1 -17892.046,E2 -17892.046} C_VEL
LIN {X 0,Y 295.962,Z 205.509,A -85,B 0,C 180,E1 -17893.223,E2 -17893.223} C_VEL
LIN {X 0,Y 291.6,Z 314.578,A -85,B 0,C 180,E1 -17895.875,E2 -17895.875} C_VEL
LIN {X 0,Y 290.447,Z 330.204,A -85,B 0,C 180,E1 -17896.532,E2 -17896.532} C_VEL
LIN {X 0,Y 289.019,Z 344.047,A -85,B 0,C 180,E1 -17897.358,E2 -17897.358} C_VEL
LIN {X 0,Y 287.002,Z 358.89,A -85,B 0,C 180,E1 -17898.526,E2 -17898.526} C_VEL
LIN {X 0,Y 284.624,Z 373.73,A -85,B 0,C 180,E1 -17900.046,E2 -17900.046} C_VEL
LIN {X 0,Y 282.301,Z 385.939,A -85,B 0,C 180,E1 -17901.589,E2 -17901.589} C_VEL
LIN {X 0,Y 279.764,Z 398.322,A -85,B 0,C 180,E1 -17903.508,E2 -17903.508} C_VEL
LIN {X 0,Y 277.353,Z 409.587,A -85,B 0,C 180,E1 -17905.64,E2 -17905.64} C_VEL
LIN {X 0,Y 275.212,Z 419.086,A -85,B 0,C 180,E1 -17907.804,E2 -17907.804} C_VEL
LIN {X 0,Y 273.146,Z 428.427,A -85,B 0,C 180,E1 -17910.368,E2 -17910.368} C_VEL
LIN {X 0,Y 271.459,Z 436.205,A -85,B 0,C 180,E1 -17912.967,E2 -17912.967} C_VEL
LIN {X 0,Y 270.012,Z 443.479,A -85,B 0,C 180,E1 -17915.976,E2 -17915.976} C_VEL
LIN {X 0,Y 269.021,Z 449.223,A -85,B 0,C 180,E1 -17919.018,E2 -17919.018} C_VEL
LIN {X 0,Y 268.352,Z 453.586,A -85,B 0,C 180,E1 -17922.093,E2 -17922.093} C_VEL
LIN {X 0,Y 267.966,Z 456.66,A -85,B 0,C 180,E1 -17925.204,E2 -17925.204} C_VEL
LIN {X 0,Y 267.859,Z 458.489,A -85,B 0,C 180,E1 -17928.351,E2 -17928.351} C_VEL
LIN {X 0,Y 267.923,Z 459.077,A -85,B 0,C 180,E1 -17931.545,E2 -17931.545} C_VEL
LIN {X 0,Y 268.284,Z 458.384,A -85,B 0,C 180,E1 -17934.78,E2 -17934.78} C_VEL
LIN {X 0,Y 269.029,Z 456.354,A -85,B 0,C 180,E1 -17938.048,E2 -17938.048} C_VEL
LIN {X 0,Y 270.274,Z 452.904,A -85,B 0,C 180,E1 -17941.336,E2 -17941.336} C_VEL
LIN {X 0,Y 272.087,Z 447.921,A -85,B 0,C 180,E1 -17944.628,E2 -17944.628} C_VEL
LIN {X 0,Y 274.16,Z 442.437,A -85,B 0,C 180,E1 -17947.374,E2 -17947.374} C_VEL
LIN {X 0,Y 276.665,Z 435.891,A -85,B 0,C 180,E1 -17949.992,E2 -17949.992} C_VEL
LIN {X 0,Y 279.771,Z 427.513,A -85,B 0,C 180,E1 -17952.707,E2 -17952.707} C_VEL
LIN {X 0,Y 283.032,Z 418.608,A -85,B 0,C 180,E1 -17955.046,E2 -17955.046} C_VEL
LIN {X 0,Y 286.754,Z 407.963,A -85,B 0,C 180,E1 -17957.329,E2 -17957.329} C_VEL
LIN {X 0,Y 290.486,Z 396.197,A -85,B 0,C 180,E1 -17959.387,E2 -17959.387} C_VEL
LIN {X 0,Y 294.223,Z 383.349,A -85,B 0,C 180,E1 -17961.196,E2 -17961.196} C_VEL
LIN {X 0,Y 297.387,Z 370.911,A -85,B 0,C 180,E1 -17962.62,E2 -17962.62} C_VEL
LIN {X 0,Y 300.336,Z 357.19,A -85,B 0,C 180,E1 -17963.885,E2 -17963.885} C_VEL
LIN {X 0,Y 302.828,Z 343.137,A -85,B 0,C 180,E1 -17964.892,E2 -17964.892} C_VEL
LIN {X 0,Y 304.611,Z 330.76,A -85,B 0,C 180,E1 -17965.57,E2 -17965.57} C_VEL
LIN {X 0,Y 306.246,Z 314.927,A -85,B 0,C 180,E1 -17966.181,E2 -17966.181} C_VEL
LIN {X 0,Y 311.361,Z 216.376,A -85,B 0,C 180,E1 -17968.534,E2 -17968.534} C_VEL
LIN {X 0,Y 309.167,Z 211.899,A -85,B 0,C 180,E1 -17969.101,E2 -17969.101} C_VEL
LIN {X 0,Y 306.552,Z 207.937,A -85,B 0,C 180,E1 -17969.752,E2 -17969.752} C_VEL
LIN {X 0,Y 301.318,Z 202.894,A -85,B 0,C 180,E1 -17971.02,E2 -17971.02} C_VEL
LIN {X 0,Y 295.054,Z 197.072,A -85,B 0,C 180,E1 -17972.639,E2 -17972.639} C_VEL
LIN {X 0,Y 293.287,Z 194.642,A -85,B 0,C 180,E1 -17973.148,E2 -17973.148} C_VEL
LIN {X 0,Y 286.199,Z 183.388,A -85,B 0,C 180,E1 -17975.395,E2 -17975.395} C_VEL
LIN {X 0,Y 281.693,Z 177.356,A -85,B 0,C 180,E1 -17976.912,E2 -17976.912} C_VEL
LIN {X 0,Y 278.913,Z 173.642,A -85,B 0,C 180,E1 -17977.913,E2 -17977.913} C_VEL
LIN {X 0,Y 275.463,Z 169.176,A -85,B 0,C 180,E1 -17979.216,E2 -17979.216} C_VEL
LIN {X 0,Y 272.708,Z 165.929,A -85,B 0,C 180,E1 -17980.305,E2 -17980.305} C_VEL
LIN {X 0,Y 271.697,Z 164.282,A -85,B 0,C 180,E1 -17980.742,E2 -17980.742} C_VEL
LIN {X 0,Y 269.06,Z 161.755,A -85,B 0,C 180,E1 -17981.831,E2 -17981.831} C_VEL
LIN {X 0,Y 267.425,Z 158.933,A -85,B 0,C 180,E1 -17982.605,E2 -17982.605} C_VEL
LIN {X 0,Y 264.921,Z 157.064,A -85,B 0,C 180,E1 -17983.724,E2 -17983.724} C_VEL
LIN {X 0,Y 263.646,Z 154.718,A -85,B 0,C 180,E1 -17984.407,E2 -17984.407} C_VEL
LIN {X 0,Y 263.33,Z 153.302,A -85,B 0,C 180,E1 -17984.669,E2 -17984.669} C_VEL
LIN {X 0,Y 263.374,Z 153.301,A -85,B 0,C 180,E1 -17989.234,E2 -17989.234} C_VEL
LIN {X 0,Y 263.573,Z 153.275,A -85,B 0,C 180,E1 -17992.338,E2 -17992.338} C_VEL
LIN {X 0,Y 263.75,Z 153.246,A -85,B 0,C 180,E1 -17998.472,E2 -17998.472} C_VEL
LIN {X 0,Y 263.75,Z 153.246,A -85,B 0,C 180,E1 -18001.526,E2 -18001.526} C_VEL
LIN {X 0,Y 263.527,Z 153.281,A -85,B 0,C 180,E1 -18007.662,E2 -18007.662} C_VEL
LIN {X 0,Y 263.349,Z 153.308,A -85,B 0,C 180,E1 -18010.766,E2 -18010.766} C_VEL
LIN {X 0,Y 263.35,Z 153.297,A -85,B 0,C 180,E1 -18015.477,E2 -18015.477} C_VEL
LIN {X 0,Y 263.262,Z 153.308,A -85,B 0,C 180,E1 -18020.306,E2 -18020.306} C_VEL
LIN {X 0,Y 263.207,Z 153.32,A -85,B 0,C 180,E1 -18025.291,E2 -18025.291} C_VEL
LIN {X 0,Y 263.164,Z 153.323,A -85,B 0,C 180,E1 -18028.731,E2 -18028.731} C_VEL
LIN {X 0,Y 263.179,Z 153.508,A -85,B 0,C 180,E1 -18031.42,E2 -18031.42} C_VEL
LIN {X 0,Y 265.24,Z 158.956,A -85,B 0,C 180,E1 -18035.182,E2 -18035.182} C_VEL
LIN {X 0,Y 269,Z 164.121,A -85,B 0,C 180,E1 -18036.934,E2 -18036.934} C_VEL
LIN {X 0,Y 270.513,Z 165.968,A -85,B 0,C 180,E1 -18037.584,E2 -18037.584} C_VEL
LIN {X 0,Y 273.985,Z 170.79,A -85,B 0,C 180,E1 -18039.034,E2 -18039.034} C_VEL
LIN {X 0,Y 279.46,Z 178.824,A -85,B 0,C 180,E1 -18041.154,E2 -18041.154} C_VEL
LIN {X 0,Y 283.255,Z 184.525,A -85,B 0,C 180,E1 -18042.508,E2 -18042.508} C_VEL
LIN {X 0,Y 289.107,Z 193.939,A -85,B 0,C 180,E1 -18044.461,E2 -18044.461} C_VEL
LIN {X 0,Y 296.243,Z 206.513,A -85,B 0,C 180,E1 -18046.653,E2 -18046.653} C_VEL
LIN {X 0,Y 302.474,Z 219.241,A -85,B 0,C 180,E1 -18048.471,E2 -18048.471} C_VEL
LIN {X 0,Y 305.968,Z 227.128,A -85,B 0,C 180,E1 -18049.455,E2 -18049.455} C_VEL
LIN {X 0,Y 300.575,Z 327.352,A -85,B 0,C 180,E1 -18051.872,E2 -18051.872} C_VEL
LIN {X 0,Y 298.754,Z 343.042,A -85,B 0,C 180,E1 -18052.452,E2 -18052.452} C_VEL
LIN {X 0,Y 296.191,Z 358.624,A -85,B 0,C 180,E1 -18053.299,E2 -18053.299} C_VEL
LIN {X 0,Y 293.44,Z 372.092,A -85,B 0,C 180,E1 -18054.283,E2 -18054.283} C_VEL
LIN {X 0,Y 289.902,Z 386.542,A -85,B 0,C 180,E1 -18055.646,E2 -18055.646} C_VEL
LIN {X 0,Y 286.129,Z 400.125,A -85,B 0,C 180,E1 -18057.292,E2 -18057.292} C_VEL
LIN {X 0,Y 282.226,Z 412.263,A -85,B 0,C 180,E1 -18059.096,E2 -18059.096} C_VEL
LIN {X 0,Y 278.141,Z 424.195,A -85,B 0,C 180,E1 -18061.309,E2 -18061.309} C_VEL
LIN {X 0,Y 274.565,Z 433.772,A -85,B 0,C 180,E1 -18063.471,E2 -18063.471} C_VEL
LIN {X 0,Y 271.309,Z 442.629,A -85,B 0,C 180,E1 -18065.922,E2 -18065.922} C_VEL
LIN {X 0,Y 268.323,Z 450.288,A -85,B 0,C 180,E1 -18068.489,E2 -18068.489} C_VEL
LIN {X 0,Y 265.592,Z 457.484,A -85,B 0,C 180,E1 -18071.486,E2 -18071.486} C_VEL
LIN {X 0,Y 263.536,Z 463.217,A -85,B 0,C 180,E1 -18074.534,E2 -18074.534} C_VEL
LIN {X 0,Y 262.179,Z 467.64,A -85,B 0,C 180,E1 -18077.617,E2 -18077.617} C_VEL
LIN {X 0,Y 261.4,Z 470.855,A -85,B 0,C 180,E1 -18080.717,E2 -18080.717} C_VEL
LIN {X 0,Y 261.045,Z 472.858,A -85,B 0,C 180,E1 -18083.818,E2 -18083.818} C_VEL
LIN {X 0,Y 261.034,Z 473.716,A -85,B 0,C 180,E1 -18086.914,E2 -18086.914} C_VEL
LIN {X 0,Y 261.125,Z 473.446,A -85,B 0,C 180,E1 -18090.001,E2 -18090.001} C_VEL
LIN {X 0,Y 261.081,Z 472.017,A -85,B 0,C 180,E1 -18093.087,E2 -18093.087} C_VEL
LIN {X 0,Y 261.136,Z 469.383,A -85,B 0,C 180,E1 -18096.181,E2 -18096.181} C_VEL
LIN {X 0,Y 261.374,Z 465.44,A -85,B 0,C 180,E1 -18099.285,E2 -18099.285} C_VEL
LIN {X 0,Y 262.004,Z 460.125,A -85,B 0,C 180,E1 -18102.392,E2 -18102.392} C_VEL
LIN {X 0,Y 263.118,Z 453.303,A -85,B 0,C 180,E1 -18105.493,E2 -18105.493} C_VEL
LIN {X 0,Y 264.626,Z 445.928,A -85,B 0,C 180,E1 -18108.184,E2 -18108.184} C_VEL
LIN {X 0,Y 266.595,Z 437.045,A -85,B 0,C 180,E1 -18110.849,E2 -18110.849} C_VEL
LIN {X 0,Y 268.98,Z 426.765,A -85,B 0,C 180,E1 -18113.376,E2 -18113.376} C_VEL
LIN {X 0,Y 271.52,Z 415.289,A -85,B 0,C 180,E1 -18115.694,E2 -18115.694} C_VEL
LIN {X 0,Y 274.181,Z 403.218,A -85,B 0,C 180,E1 -18117.685,E2 -18117.685} C_VEL
LIN {X 0,Y 276.549,Z 391.417,A -85,B 0,C 180,E1 -18119.289,E2 -18119.289} C_VEL
LIN {X 0,Y 279.021,Z 378.086,A -85,B 0,C 180,E1 -18120.76,E2 -18120.76} C_VEL
LIN {X 0,Y 281.218,Z 364.249,A -85,B 0,C 180,E1 -18121.973,E2 -18121.973} C_VEL
LIN {X 0,Y 283.066,Z 349.767,A -85,B 0,C 180,E1 -18122.95,E2 -18122.95} C_VEL
LIN {X 0,Y 284.55,Z 335.225,A -85,B 0,C 180,E1 -18123.655,E2 -18123.655} C_VEL
LIN {X 0,Y 285.526,Z 319.19,A -85,B 0,C 180,E1 -18124.161,E2 -18124.161} C_VEL
LIN {X 0,Y 289.402,Z 220.066,A -85,B 0,C 180,E1 -18126.592,E2 -18126.592} C_VEL
LIN {X 0,Y 287.838,Z 210.828,A -85,B 0,C 180,E1 -18127.05,E2 -18127.05} C_VEL
LIN {X 0,Y 279.67,Z 190.938,A -85,B 0,C 180,E1 -18128.683,E2 -18128.683} C_VEL
LIN {X 0,Y 271.417,Z 173.095,A -85,B 0,C 180,E1 -18130.386,E2 -18130.386} C_VEL
LIN {X 0,Y 265.329,Z 161.091,A -85,B 0,C 180,E1 -18131.723,E2 -18131.723} C_VEL
LIN {X 0,Y 263.113,Z 153.339,A -85,B 0,C 180,E1 -18134.465,E2 -18134.465} C_VEL
LIN {X 0,Y 263.126,Z 153.338,A -85,B 0,C 180,E1 -18138.407,E2 -18138.407} C_VEL
LIN {X 0,Y 263.184,Z 153.329,A -85,B 0,C 180,E1 -18143.238,E2 -18143.238} C_VEL
LIN {X 0,Y 263.13,Z 153.33,A -85,B 0,C 180,E1 -18147.712,E2 -18147.712} C_VEL
LIN {X 0,Y 263.15,Z 153.3,A -85,B 0,C 180,E1 -18151.806,E2 -18151.806} C_VEL
LIN {X 0,Y 263.192,Z 153.319,A -85,B 0,C 180,E1 -18155.219,E2 -18155.219} C_VEL
LIN {X 0,Y 263.242,Z 153.317,A -85,B 0,C 180,E1 -18159.692,E2 -18159.692} C_VEL
LIN {X 0,Y 263.327,Z 153.305,A -85,B 0,C 180,E1 -18164.521,E2 -18164.521} C_VEL
LIN {X 0,Y 263.354,Z 153.305,A -85,B 0,C 180,E1 -18169.234,E2 -18169.234} C_VEL
LIN {X 0,Y 263.53,Z 153.276,A -85,B 0,C 180,E1 -18172.338,E2 -18172.338} C_VEL
LIN {X 0,Y 263.738,Z 153.222,A -85,B 0,C 180,E1 -18178.474,E2 -18178.474} C_VEL
LIN {X 0,Y 263.736,Z 153.235,A -85,B 0,C 180,E1 -18181.528,E2 -18181.528} C_VEL
LIN {X 0,Y 263.531,Z 153.255,A -85,B 0,C 180,E1 -18187.663,E2 -18187.663} C_VEL
LIN {X 0,Y 263.331,Z 153.273,A -85,B 0,C 180,E1 -18190.768,E2 -18190.768} C_VEL
LIN {X 0,Y 263.293,Z 153.311,A -85,B 0,C 180,E1 -18195.482,E2 -18195.482} C_VEL
LIN {X 0,Y 263.203,Z 153.322,A -85,B 0,C 180,E1 -18200.312,E2 -18200.312} C_VEL
LIN {X 0,Y 263.124,Z 153.334,A -85,B 0,C 180,E1 -18205.301,E2 -18205.301} C_VEL
LIN {X 0,Y 263.122,Z 153.298,A -85,B 0,C 180,E1 -18208.737,E2 -18208.737} C_VEL
LIN {X 0,Y 263.131,Z 153.325,A -85,B 0,C 180,E1 -18212.289,E2 -18212.289} C_VEL
LIN {X 0,Y 263.179,Z 153.303,A -85,B 0,C 180,E1 -18216.761,E2 -18216.761} C_VEL
LIN {X 0,Y 263.096,Z 153.317,A -85,B 0,C 180,E1 -18219.875,E2 -18219.875} C_VEL
LIN {X 0,Y 263.081,Z 153.328,A -85,B 0,C 180,E1 -18223.994,E2 -18223.994} C_VEL
LIN {X 0,Y 263.081,Z 153.335,A -85,B 0,C 180,E1 -18228.097,E2 -18228.097} C_VEL
LIN {X 0,Y 263.108,Z 153.317,A -85,B 0,C 180,E1 -18232.093,E2 -18232.093} C_VEL
LIN {X 0,Y 263.156,Z 153.327,A -85,B 0,C 180,E1 -18235.885,E2 -18235.885} C_VEL
LIN {X 0,Y 263.131,Z 153.336,A -85,B 0,C 180,E1 -18239.503,E2 -18239.503} C_VEL
LIN {X 0,Y 263.144,Z 153.332,A -85,B 0,C 180,E1 -18242.996,E2 -18242.996} C_VEL
LIN {X 0,Y 263.179,Z 153.379,A -85,B 0,C 180,E1 -18247.189,E2 -18247.189} C_VEL
LIN {X 0,Y 264.037,Z 155.969,A -85,B 0,C 180,E1 -18247.411,E2 -18247.411} C_VEL
LIN {X 0,Y 265.751,Z 158.485,A -85,B 0,C 180,E1 -18247.761,E2 -18247.761} C_VEL
LIN {X 0,Y 273.721,Z 171.921,A -85,B 0,C 180,E1 -18249.378,E2 -18249.378} C_VEL
LIN {X 0,Y 279.222,Z 182.394,A -85,B 0,C 180,E1 -18250.463,E2 -18250.463} C_VEL
LIN {X 0,Y 287.677,Z 201.895,A -85,B 0,C 180,E1 -18252.138,E2 -18252.138} C_VEL
LIN {X 0,Y 289.779,Z 207.6,A -85,B 0,C 180,E1 -18252.56,E2 -18252.56} C_VEL
LIN {X 0,Y 285.376,Z 314.331,A -85,B 0,C 180,E1 -18255.196,E2 -18255.196} C_VEL
LIN {X 0,Y 284.175,Z 330.129,A -85,B 0,C 180,E1 -18255.864,E2 -18255.864} C_VEL
LIN {X 0,Y 282.706,Z 344.016,A -85,B 0,C 180,E1 -18256.705,E2 -18256.705} C_VEL
LIN {X 0,Y 280.758,Z 358.022,A -85,B 0,C 180,E1 -18257.817,E2 -18257.817} C_VEL
LIN {X 0,Y 278.446,Z 372.305,A -85,B 0,C 180,E1 -18259.271,E2 -18259.271} C_VEL
LIN {X 0,Y 276.056,Z 384.738,A -85,B 0,C 180,E1 -18260.844,E2 -18260.844} C_VEL
LIN {X 0,Y 273.612,Z 396.3,A -85,B 0,C 180,E1 -18262.621,E2 -18262.621} C_VEL
LIN {X 0,Y 271.022,Z 407.939,A -85,B 0,C 180,E1 -18264.792,E2 -18264.792} C_VEL
LIN {X 0,Y 268.699,Z 417.753,A -85,B 0,C 180,E1 -18267.001,E2 -18267.001} C_VEL
LIN {X 0,Y 266.825,Z 426.211,A -85,B 0,C 180,E1 -18269.279,E2 -18269.279} C_VEL
LIN {X 0,Y 264.939,Z 434.333,A -85,B 0,C 180,E1 -18271.9,E2 -18271.9} C_VEL
LIN {X 0,Y 263.513,Z 441.13,A -85,B 0,C 180,E1 -18274.589,E2 -18274.589} C_VEL
LIN {X 0,Y 262.292,Z 447.436,A -85,B 0,C 180,E1 -18277.699,E2 -18277.699} C_VEL
LIN {X 0,Y 261.49,Z 452.301,A -85,B 0,C 180,E1 -18280.844,E2 -18280.844} C_VEL
LIN {X 0,Y 260.972,Z 456.002,A -85,B 0,C 180,E1 -18284.188,E2 -18284.188} C_VEL
LIN {X 0,Y 260.747,Z 458.139,A -85,B 0,C 180,E1 -18287.246,E2 -18287.246} C_VEL
LIN {X 0,Y 260.79,Z 458.989,A -85,B 0,C 180,E1 -18289.4,E2 -18289.4} C_VEL
LIN {X 0,Y 260.884,Z 459.243,A -85,B 0,C 180,E1 -18292.157,E2 -18292.157} C_VEL
LIN {X 0,Y 261.321,Z 458.384,A -85,B 0,C 180,E1 -18295.486,E2 -18295.486} C_VEL
LIN {X 0,Y 262.175,Z 456.185,A -85,B 0,C 180,E1 -18298.849,E2 -18298.849} C_VEL
LIN {X 0,Y 263.58,Z 452.558,A -85,B 0,C 180,E1 -18302.226,E2 -18302.226} C_VEL
LIN {X 0,Y 265.62,Z 447.385,A -85,B 0,C 180,E1 -18305.597,E2 -18305.597} C_VEL
LIN {X 0,Y 267.897,Z 441.794,A -85,B 0,C 180,E1 -18308.388,E2 -18308.388} C_VEL
LIN {X 0,Y 270.76,Z 434.765,A -85,B 0,C 180,E1 -18311.171,E2 -18311.171} C_VEL
LIN {X 0,Y 274.008,Z 426.423,A -85,B 0,C 180,E1 -18313.829,E2 -18313.829} C_VEL
LIN {X 0,Y 277.514,Z 417.253,A -85,B 0,C 180,E1 -18316.199,E2 -18316.199} C_VEL
LIN {X 0,Y 281.474,Z 406.313,A -85,B 0,C 180,E1 -18318.508,E2 -18318.508} C_VEL
LIN {X 0,Y 285.415,Z 394.213,A -85,B 0,C 180,E1 -18320.585,E2 -18320.585} C_VEL
LIN {X 0,Y 289.242,Z 381.403,A -85,B 0,C 180,E1 -18322.344,E2 -18322.344} C_VEL
LIN {X 0,Y 292.671,Z 367.873,A -85,B 0,C 180,E1 -18323.847,E2 -18323.847} C_VEL
LIN {X 0,Y 295.529,Z 354.736,A -85,B 0,C 180,E1 -18324.995,E2 -18324.995} C_VEL
LIN {X 0,Y 297.943,Z 340.912,A -85,B 0,C 180,E1 -18325.949,E2 -18325.949} C_VEL
LIN {X 0,Y 299.92,Z 326.681,A -85,B 0,C 180,E1 -18326.671,E2 -18326.671} C_VEL
LIN {X 0,Y 301.323,Z 311.06,A -85,B 0,C 180,E1 -18327.221,E2 -18327.221} C_VEL
LIN {X 0,Y 306.349,Z 219.212,A -85,B 0,C 180,E1 -18329.402,E2 -18329.402} C_VEL
LIN {X 0,Y 299.99,Z 206.391,A -85,B 0,C 180,E1 -18331.181,E2 -18331.181} C_VEL
LIN {X 0,Y 293.528,Z 195.064,A -85,B 0,C 180,E1 -18333.075,E2 -18333.075} C_VEL
LIN {X 0,Y 293.287,Z 194.642,A -85,B 0,C 180,E1 -18333.148,E2 -18333.148} C_VEL
LIN {X 0,Y 291.415,Z 192.509,A -85,B 0,C 180,E1 -18333.685,E2 -18333.685} C_VEL
LIN {X 0,Y 287.714,Z 190.455,A -85,B 0,C 180,E1 -18334.699,E2 -18334.699} C_VEL
LIN {X 0,Y 283.189,Z 188.427,A -85,B 0,C 180,E1 -18335.998,E2 -18335.998} C_VEL
LIN {X 0,Y 281.841,Z 187.372,A -85,B 0,C 180,E1 -18336.422,E2 -18336.422} C_VEL
LIN {X 0,Y 276.325,Z 179.74,A -85,B 0,C 180,E1 -18338.431,E2 -18338.431} C_VEL
LIN {X 0,Y 272.621,Z 175.049,A -85,B 0,C 180,E1 -18339.871,E2 -18339.871} C_VEL
LIN {X 0,Y 269.633,Z 171.095,A -85,B 0,C 180,E1 -18341.12,E2 -18341.12} C_VEL
LIN {X 0,Y 266.284,Z 167.294,A -85,B 0,C 180,E1 -18342.578,E2 -18342.578} C_VEL
LIN {X 0,Y 265.024,Z 165.324,A -85,B 0,C 180,E1 -18343.194,E2 -18343.194} C_VEL
LIN {X 0,Y 262.538,Z 163.053,A -85,B 0,C 180,E1 -18344.374,E2 -18344.374} C_VEL
LIN {X 0,Y 260.753,Z 159.922,A -85,B 0,C 180,E1 -18345.363,E2 -18345.363} C_VEL
LIN {X 0,Y 258.127,Z 158.163,A -85,B 0,C 180,E1 -18346.718,E2 -18346.718} C_VEL
LIN {X 0,Y 256.766,Z 155.96,A -85,B 0,C 180,E1 -18347.552,E2 -18347.552} C_VEL
LIN {X 0,Y 256.286,Z 154.177,A -85,B 0,C 180,E1 -18347.98,E2 -18347.98} C_VEL
LIN {X 0,Y 256.497,Z 154.153,A -85,B 0,C 180,E1 -18350.537,E2 -18350.537} C_VEL
LIN {X 0,Y 256.487,Z 154.154,A -85,B 0,C 180,E1 -18353.707,E2 -18353.707} C_VEL
LIN {X 0,Y 256.713,Z 154.123,A -85,B 0,C 180,E1 -18358.431,E2 -18358.431} C_VEL
LIN {X 0,Y 256.713,Z 154.122,A -85,B 0,C 180,E1 -18361.568,E2 -18361.568} C_VEL
LIN {X 0,Y 256.46,Z 154.158,A -85,B 0,C 180,E1 -18366.293,E2 -18366.293} C_VEL
LIN {X 0,Y 256.425,Z 154.159,A -85,B 0,C 180,E1 -18369.464,E2 -18369.464} C_VEL
LIN {X 0,Y 256.255,Z 154.19,A -85,B 0,C 180,E1 -18374.29,E2 -18374.29} C_VEL
LIN {X 0,Y 256.21,Z 154.193,A -85,B 0,C 180,E1 -18377.561,E2 -18377.561} C_VEL
LIN {X 0,Y 256.156,Z 154.202,A -85,B 0,C 180,E1 -18381.12,E2 -18381.12} C_VEL
LIN {X 0,Y 256.187,Z 154.195,A -85,B 0,C 180,E1 -18385.138,E2 -18385.138} C_VEL
LIN {X 0,Y 256.149,Z 154.322,A -85,B 0,C 180,E1 -18388.441,E2 -18388.441} C_VEL
LIN {X 0,Y 257.649,Z 158.358,A -85,B 0,C 180,E1 -18391.719,E2 -18391.719} C_VEL
LIN {X 0,Y 260.485,Z 162.392,A -85,B 0,C 180,E1 -18393.334,E2 -18393.334} C_VEL
LIN {X 0,Y 263.622,Z 166.091,A -85,B 0,C 180,E1 -18394.933,E2 -18394.933} C_VEL
LIN {X 0,Y 266.741,Z 170.43,A -85,B 0,C 180,E1 -18396.431,E2 -18396.431} C_VEL
LIN {X 0,Y 268.282,Z 172.528,A -85,B 0,C 180,E1 -18397.123,E2 -18397.123} C_VEL
LIN {X 0,Y 273.004,Z 179.185,A -85,B 0,C 180,E1 -18399.126,E2 -18399.126} C_VEL
LIN {X 0,Y 276.689,Z 184.794,A -85,B 0,C 180,E1 -18400.584,E2 -18400.584} C_VEL
LIN {X 0,Y 280.708,Z 191.02,A -85,B 0,C 180,E1 -18402.076,E2 -18402.076} C_VEL
LIN {X 0,Y 286.505,Z 200.673,A -85,B 0,C 180,E1 -18404.071,E2 -18404.071} C_VEL
LIN {X 0,Y 292.499,Z 211.478,A -85,B 0,C 180,E1 -18405.977,E2 -18405.977} C_VEL
LIN {X 0,Y 298.829,Z 224.63,A -85,B 0,C 180,E1 -18407.892,E2 -18407.892} C_VEL
LIN {X 0,Y 301.022,Z 229.746,A -85,B 0,C 180,E1 -18408.541,E2 -18408.541} C_VEL
LIN {X 0,Y 295.478,Z 327.507,A -85,B 0,C 180,E1 -18410.928,E2 -18410.928} C_VEL
LIN {X 0,Y 293.564,Z 343.058,A -85,B 0,C 180,E1 -18411.505,E2 -18411.505} C_VEL
LIN {X 0,Y 291.049,Z 358.022,A -85,B 0,C 180,E1 -18412.322,E2 -18412.322} C_VEL
LIN {X 0,Y 288.201,Z 371.542,A -85,B 0,C 180,E1 -18413.313,E2 -18413.313} C_VEL
LIN {X 0,Y 284.463,Z 386.338,A -85,B 0,C 180,E1 -18414.716,E2 -18414.716} C_VEL
LIN {X 0,Y 280.665,Z 399.705,A -85,B 0,C 180,E1 -18416.357,E2 -18416.357} C_VEL
LIN {X 0,Y 276.559,Z 411.879,A -85,B 0,C 180,E1 -18418.177,E2 -18418.177} C_VEL
LIN {X 0,Y 272.588,Z 422.994,A -85,B 0,C 180,E1 -18420.244,E2 -18420.244} C_VEL
LIN {X 0,Y 268.219,Z 434.155,A -85,B 0,C 180,E1 -18422.792,E2 -18422.792} C_VEL
LIN {X 0,Y 264.346,Z 444.08,A -85,B 0,C 180,E1 -18425.664,E2 -18425.664} C_VEL
LIN {X 0,Y 260.931,Z 452.421,A -85,B 0,C 180,E1 -18428.678,E2 -18428.678} C_VEL
LIN {X 0,Y 258.189,Z 459.168,A -85,B 0,C 180,E1 -18431.758,E2 -18431.758} C_VEL
LIN {X 0,Y 256.243,Z 464.501,A -85,B 0,C 180,E1 -18434.897,E2 -18434.897} C_VEL
LIN {X 0,Y 255.208,Z 467.611,A -85,B 0,C 180,E1 -18437.274,E2 -18437.274} C_VEL
LIN {X 0,Y 254.343,Z 470.759,A -85,B 0,C 180,E1 -18440.457,E2 -18440.457} C_VEL
LIN {X 0,Y 253.958,Z 472.731,A -85,B 0,C 180,E1 -18443.645,E2 -18443.645} C_VEL
LIN {X 0,Y 253.933,Z 473.53,A -85,B 0,C 180,E1 -18446.827,E2 -18446.827} C_VEL
LIN {X 0,Y 254.053,Z 473.204,A -85,B 0,C 180,E1 -18450.001,E2 -18450.001} C_VEL
LIN {X 0,Y 253.978,Z 471.715,A -85,B 0,C 180,E1 -18453.173,E2 -18453.173} C_VEL
LIN {X 0,Y 254.041,Z 469.026,A -85,B 0,C 180,E1 -18456.354,E2 -18456.354} C_VEL
LIN {X 0,Y 254.311,Z 465.043,A -85,B 0,C 180,E1 -18459.545,E2 -18459.545} C_VEL
LIN {X 0,Y 255.019,Z 459.663,A -85,B 0,C 180,E1 -18462.737,E2 -18462.737} C_VEL
LIN {X 0,Y 256.178,Z 452.766,A -85,B 0,C 180,E1 -18465.923,E2 -18465.923} C_VEL
LIN {X 0,Y 257.778,Z 445.309,A -85,B 0,C 180,E1 -18468.685,E2 -18468.685} C_VEL
LIN {X 0,Y 259.879,Z 436.332,A -85,B 0,C 180,E1 -18471.414,E2 -18471.414} C_VEL
LIN {X 0,Y 262.083,Z 427.167,A -85,B 0,C 180,E1 -18473.719,E2 -18473.719} C_VEL
LIN {X 0,Y 264.582,Z 416.321,A -85,B 0,C 180,E1 -18475.995,E2 -18475.995} C_VEL
LIN {X 0,Y 267.277,Z 404.483,A -85,B 0,C 180,E1 -18478.036,E2 -18478.036} C_VEL
LIN {X 0,Y 269.707,Z 392.987,A -85,B 0,C 180,E1 -18479.677,E2 -18479.677} C_VEL
LIN {X 0,Y 272.338,Z 379.607,A -85,B 0,C 180,E1 -18481.223,E2 -18481.223} C_VEL
LIN {X 0,Y 274.627,Z 365.67,A -85,B 0,C 180,E1 -18482.509,E2 -18482.509} C_VEL
LIN {X 0,Y 276.706,Z 350.226,A -85,B 0,C 180,E1 -18483.589,E2 -18483.589} C_VEL
LIN {X 0,Y 278.312,Z 334.858,A -85,B 0,C 180,E1 -18484.35,E2 -18484.35} C_VEL
LIN {X 0,Y 279.331,Z 318.745,A -85,B 0,C 180,E1 -18484.863,E2 -18484.863} C_VEL
LIN {X 0,Y 283.276,Z 221.169,A -85,B 0,C 180,E1 -18487.302,E2 -18487.302} C_VEL
LIN {X 0,Y 282.004,Z 213.368,A -85,B 0,C 180,E1 -18487.697,E2 -18487.697} C_VEL
LIN {X 0,Y 273.752,Z 193.22,A -85,B 0,C 180,E1 -18489.413,E2 -18489.413} C_VEL
LIN {X 0,Y 265.932,Z 176.338,A -85,B 0,C 180,E1 -18491.087,E2 -18491.087} C_VEL
LIN {X 0,Y 259.477,Z 164.055,A -85,B 0,C 180,E1 -18492.505,E2 -18492.505} C_VEL
LIN {X 0,Y 257.965,Z 160.894,A -85,B 0,C 180,E1 -18492.888,E2 -18492.888} C_VEL
LIN {X 0,Y 256.056,Z 154.22,A -85,B 0,C 180,E1 -18495.366,E2 -18495.366} C_VEL
LIN {X 0,Y 256.057,Z 154.22,A -85,B 0,C 180,E1 -18498.798,E2 -18498.798} C_VEL
LIN {X 0,Y 256.132,Z 154.205,A -85,B 0,C 180,E1 -18502.868,E2 -18502.868} C_VEL
LIN {X 0,Y 256.068,Z 154.21,A -85,B 0,C 180,E1 -18506.708,E2 -18506.708} C_VEL
LIN {X 0,Y 256.057,Z 154.2,A -85,B 0,C 180,E1 -18510.394,E2 -18510.394} C_VEL
LIN {X 0,Y 256.135,Z 154.195,A -85,B 0,C 180,E1 -18514.889,E2 -18514.889} C_VEL
LIN {X 0,Y 256.151,Z 154.195,A -85,B 0,C 180,E1 -18519.104,E2 -18519.104} C_VEL
LIN {X 0,Y 256.262,Z 154.182,A -85,B 0,C 180,E1 -18524.083,E2 -18524.083} C_VEL
LIN {X 0,Y 256.295,Z 154.182,A -85,B 0,C 180,E1 -18528.934,E2 -18528.934} C_VEL
LIN {X 0,Y 256.472,Z 154.155,A -85,B 0,C 180,E1 -18532.126,E2 -18532.126} C_VEL
LIN {X 0,Y 256.455,Z 154.152,A -85,B 0,C 180,E1 -18536.859,E2 -18536.859} C_VEL
LIN {X 0,Y 256.7,Z 154.098,A -85,B 0,C 180,E1 -18538.432,E2 -18538.432} C_VEL
LIN {X 0,Y 256.698,Z 154.111,A -85,B 0,C 180,E1 -18541.57,E2 -18541.57} C_VEL
LIN {X 0,Y 256.447,Z 154.149,A -85,B 0,C 180,E1 -18546.573,E2 -18546.573} C_VEL
LIN {X 0,Y 256.406,Z 154.127,A -85,B 0,C 180,E1 -18549.466,E2 -18549.466} C_VEL
LIN {X 0,Y 256.2,Z 154.195,A -85,B 0,C 180,E1 -18554.294,E2 -18554.294} C_VEL
LIN {X 0,Y 256.143,Z 154.194,A -85,B 0,C 180,E1 -18557.567,E2 -18557.567} C_VEL
LIN {X 0,Y 256.117,Z 154.202,A -85,B 0,C 180,E1 -18561.094,E2 -18561.094} C_VEL
LIN {X 0,Y 256.086,Z 154.212,A -85,B 0,C 180,E1 -18565.087,E2 -18565.087} C_VEL
LIN {X 0,Y 256.08,Z 154.175,A -85,B 0,C 180,E1 -18568.569,E2 -18568.569} C_VEL
LIN {X 0,Y 256.074,Z 154.193,A -85,B 0,C 180,E1 -18571.7,E2 -18571.7} C_VEL
LIN {X 0,Y 256.084,Z 154.205,A -85,B 0,C 180,E1 -18575.194,E2 -18575.194} C_VEL
LIN {X 0,Y 256.069,Z 154.182,A -85,B 0,C 180,E1 -18579.143,E2 -18579.143} C_VEL
LIN {X 0,Y 256.033,Z 154.212,A -85,B 0,C 180,E1 -18583.334,E2 -18583.334} C_VEL
LIN {X 0,Y 256.035,Z 154.209,A -85,B 0,C 180,E1 -18587.829,E2 -18587.829} C_VEL
LIN {X 0,Y 256.047,Z 154.206,A -85,B 0,C 180,E1 -18590.852,E2 -18590.852} C_VEL
LIN {X 0,Y 256.083,Z 154.213,A -85,B 0,C 180,E1 -18594.806,E2 -18594.806} C_VEL
LIN {X 0,Y 256.088,Z 154.203,A -85,B 0,C 180,E1 -18598.571,E2 -18598.571} C_VEL
LIN {X 0,Y 256.096,Z 154.203,A -85,B 0,C 180,E1 -18602.19,E2 -18602.19} C_VEL
LIN {X 0,Y 256.116,Z 154.265,A -85,B 0,C 180,E1 -18606.069,E2 -18606.069} C_VEL
LIN {X 0,Y 257.156,Z 157.152,A -85,B 0,C 180,E1 -18606.345,E2 -18606.345} C_VEL
LIN {X 0,Y 258.73,Z 159.36,A -85,B 0,C 180,E1 -18606.681,E2 -18606.681} C_VEL
LIN {X 0,Y 268.411,Z 175.545,A -85,B 0,C 180,E1 -18608.729,E2 -18608.729} C_VEL
LIN {X 0,Y 273.75,Z 185.711,A -85,B 0,C 180,E1 -18609.821,E2 -18609.821} C_VEL
LIN {X 0,Y 281.698,Z 204.099,A -85,B 0,C 180,E1 -18611.453,E2 -18611.453} C_VEL
LIN {X 0,Y 283.624,Z 208.884,A -85,B 0,C 180,E1 -18611.843,E2 -18611.843} C_VEL
LIN {X 0,Y 279.189,Z 313.915,A -85,B 0,C 180,E1 -18614.486,E2 -18614.486} C_VEL
LIN {X 0,Y 277.938,Z 329.971,A -85,B 0,C 180,E1 -18615.165,E2 -18615.165} C_VEL
LIN {X 0,Y 276.42,Z 343.916,A -85,B 0,C 180,E1 -18616.022,E2 -18616.022} C_VEL
LIN {X 0,Y 274.343,Z 358.457,A -85,B 0,C 180,E1 -18617.196,E2 -18617.196} C_VEL
LIN {X 0,Y 272.018,Z 372.318,A -85,B 0,C 180,E1 -18618.638,E2 -18618.638} C_VEL
LIN {X 0,Y 269.549,Z 384.784,A -85,B 0,C 180,E1 -18620.242,E2 -18620.242} C_VEL
LIN {X 0,Y 267.001,Z 396.379,A -85,B 0,C 180,E1 -18622.056,E2 -18622.056} C_VEL
LIN {X 0,Y 264.334,Z 408.04,A -85,B 0,C 180,E1 -18624.277,E2 -18624.277} C_VEL
LIN {X 0,Y 261.931,Z 417.874,A -85,B 0,C 180,E1 -18626.538,E2 -18626.538} C_VEL
LIN {X 0,Y 259.684,Z 427.482,A -85,B 0,C 180,E1 -18629.223,E2 -18629.223} C_VEL
LIN {X 0,Y 257.773,Z 435.508,A -85,B 0,C 180,E1 -18631.952,E2 -18631.952} C_VEL
LIN {X 0,Y 256.327,Z 442.177,A -85,B 0,C 180,E1 -18634.718,E2 -18634.718} C_VEL
LIN {X 0,Y 255.119,Z 448.308,A -85,B 0,C 180,E1 -18637.916,E2 -18637.916} C_VEL
LIN {X 0,Y 254.317,Z 453.026,A -85,B 0,C 180,E1 -18641.153,E2 -18641.153} C_VEL
LIN {X 0,Y 253.839,Z 456.416,A -85,B 0,C 180,E1 -18644.428,E2 -18644.428} C_VEL
LIN {X 0,Y 253.659,Z 458.546,A -85,B 0,C 180,E1 -18647.744,E2 -18647.744} C_VEL
LIN {X 0,Y 253.689,Z 459.211,A -85,B 0,C 180,E1 -18649.623,E2 -18649.623} C_VEL
LIN {X 0,Y 253.851,Z 459.411,A -85,B 0,C 180,E1 -18652.805,E2 -18652.805} C_VEL
LIN {X 0,Y 254.369,Z 458.389,A -85,B 0,C 180,E1 -18656.235,E2 -18656.235} C_VEL
LIN {X 0,Y 255.365,Z 456.019,A -85,B 0,C 180,E1 -18659.695,E2 -18659.695} C_VEL
LIN {X 0,Y 256.959,Z 452.212,A -85,B 0,C 180,E1 -18663.162,E2 -18663.162} C_VEL
LIN {X 0,Y 259.257,Z 446.85,A -85,B 0,C 180,E1 -18666.611,E2 -18666.611} C_VEL
LIN {X 0,Y 261.561,Z 441.536,A -85,B 0,C 180,E1 -18669.252,E2 -18669.252} C_VEL
LIN {X 0,Y 264.347,Z 434.998,A -85,B 0,C 180,E1 -18671.89,E2 -18671.89} C_VEL
LIN {X 0,Y 267.795,Z 426.699,A -85,B 0,C 180,E1 -18674.589,E2 -18674.589} C_VEL
LIN {X 0,Y 271.471,Z 417.561,A -85,B 0,C 180,E1 -18676.999,E2 -18676.999} C_VEL
LIN {X 0,Y 275.597,Z 406.644,A -85,B 0,C 180,E1 -18679.345,E2 -18679.345} C_VEL
LIN {X 0,Y 279.721,Z 394.581,A -85,B 0,C 180,E1 -18681.445,E2 -18681.445} C_VEL
LIN {X 0,Y 283.791,Z 381.464,A -85,B 0,C 180,E1 -18683.27,E2 -18683.27} C_VEL
LIN {X 0,Y 287.229,Z 368.316,A -85,B 0,C 180,E1 -18684.748,E2 -18684.748} C_VEL
LIN {X 0,Y 290.199,Z 355.195,A -85,B 0,C 180,E1 -18685.911,E2 -18685.911} C_VEL
LIN {X 0,Y 292.956,Z 339.751,A -85,B 0,C 180,E1 -18686.983,E2 -18686.983} C_VEL
LIN {X 0,Y 295.095,Z 324.567,A -85,B 0,C 180,E1 -18687.722,E2 -18687.722} C_VEL
LIN {X 0,Y 296.427,Z 309.216,A -85,B 0,C 180,E1 -18688.232,E2 -18688.232} C_VEL
LIN {X 0,Y 301.384,Z 221.835,A -85,B 0,C 180,E1 -18690.327,E2 -18690.327} C_VEL
LIN {X 0,Y 295.51,Z 210.138,A -85,B 0,C 180,E1 -18692.039,E2 -18692.039} C_VEL
LIN {X 0,Y 289.894,Z 200.092,A -85,B 0,C 180,E1 -18693.757,E2 -18693.757} C_VEL
LIN {X 0,Y 282.835,Z 188.637,A -85,B 0,C 180,E1 -18696.087,E2 -18696.087} C_VEL
LIN {X 0,Y 281.841,Z 187.372,A -85,B 0,C 180,E1 -18696.422,E2 -18696.422} C_VEL
LIN {X 0,Y 278.02,Z 184.316,A -85,B 0,C 180,E1 -18697.691,E2 -18697.691} C_VEL
LIN {X 0,Y 270.359,Z 179.614,A -85,B 0,C 180,E1 -18700.417,E2 -18700.417} C_VEL
LIN {X 0,Y 266.904,Z 176.821,A -85,B 0,C 180,E1 -18701.814,E2 -18701.814} C_VEL
LIN {X 0,Y 264.004,Z 173.58,A -85,B 0,C 180,E1 -18703.127,E2 -18703.127} C_VEL
LIN {X 0,Y 262.761,Z 171.689,A -85,B 0,C 180,E1 -18703.754,E2 -18703.754} C_VEL
LIN {X 0,Y 260.2,Z 169.05,A -85,B 0,C 180,E1 -18705.031,E2 -18705.031} C_VEL
LIN {X 0,Y 258.765,Z 166.568,A -85,B 0,C 180,E1 -18705.851,E2 -18705.851} C_VEL
LIN {X 0,Y 256.136,Z 164.533,A -85,B 0,C 180,E1 -18707.269,E2 -18707.269} C_VEL
LIN {X 0,Y 254.526,Z 161.877,A -85,B 0,C 180,E1 -18708.3,E2 -18708.3} C_VEL
LIN {X 0,Y 254.046,Z 160.908,A -85,B 0,C 180,E1 -18708.631,E2 -18708.631} C_VEL
LIN {X 0,Y 251.494,Z 159.246,A -85,B 0,C 180,E1 -18710.245,E2 -18710.245} C_VEL
LIN {X 0,Y 249.923,Z 156.83,A -85,B 0,C 180,E1 -18711.452,E2 -18711.452} C_VEL
LIN {X 0,Y 249.485,Z 155.026,A -85,B 0,C 180,E1 -18711.953,E2 -18711.953} C_VEL
LIN {X 0,Y 249.435,Z 155.036,A -85,B 0,C 180,E1 -18716.769,E2 -18716.769} C_VEL
LIN {X 0,Y 249.728,Z 155.004,A -85,B 0,C 180,E1 -18719.999,E2 -18719.999} C_VEL
LIN {X 0,Y 249.431,Z 155.04,A -85,B 0,C 180,E1 -18723.23,E2 -18723.23} C_VEL
LIN {X 0,Y 249.43,Z 155.035,A -85,B 0,C 180,E1 -18726.471,E2 -18726.471} C_VEL
LIN {X 0,Y 249.341,Z 155.042,A -85,B 0,C 180,E1 -18729.736,E2 -18729.736} C_VEL
LIN {X 0,Y 249.205,Z 155.067,A -85,B 0,C 180,E1 -18734.703,E2 -18734.703} C_VEL
LIN {X 0,Y 249.138,Z 155.077,A -85,B 0,C 180,E1 -18738.077,E2 -18738.077} C_VEL
LIN {X 0,Y 249.086,Z 155.084,A -85,B 0,C 180,E1 -18741.518,E2 -18741.518} C_VEL
LIN {X 0,Y 249.153,Z 155.157,A -85,B 0,C 180,E1 -18744.808,E2 -18744.808} C_VEL
LIN {X 0,Y 250.073,Z 157.891,A -85,B 0,C 180,E1 -18747.399,E2 -18747.399} C_VEL
LIN {X 0,Y 253.915,Z 162.951,A -85,B 0,C 180,E1 -18750.11,E2 -18750.11} C_VEL
LIN {X 0,Y 255.774,Z 165,A -85,B 0,C 180,E1 -18751.24,E2 -18751.24} C_VEL
LIN {X 0,Y 260.018,Z 170.625,A -85,B 0,C 180,E1 -18753.648,E2 -18753.648} C_VEL
LIN {X 0,Y 261.877,Z 173.118,A -85,B 0,C 180,E1 -18754.618,E2 -18754.618} C_VEL
LIN {X 0,Y 265.815,Z 178.618,A -85,B 0,C 180,E1 -18756.532,E2 -18756.532} C_VEL
LIN {X 0,Y 270.179,Z 184.849,A -85,B 0,C 180,E1 -18758.451,E2 -18758.451} C_VEL
LIN {X 0,Y 273.821,Z 190.546,A -85,B 0,C 180,E1 -18759.952,E2 -18759.952} C_VEL
LIN {X 0,Y 277.777,Z 196.767,A -85,B 0,C 180,E1 -18761.473,E2 -18761.473} C_VEL
LIN {X 0,Y 284.221,Z 207.826,A -85,B 0,C 180,E1 -18763.771,E2 -18763.771} C_VEL
LIN {X 0,Y 290.288,Z 219.394,A -85,B 0,C 180,E1 -18765.759,E2 -18765.759} C_VEL
LIN {X 0,Y 296.106,Z 232.217,A -85,B 0,C 180,E1 -18767.577,E2 -18767.577} C_VEL
LIN {X 0,Y 290.572,Z 326.828,A -85,B 0,C 180,E1 -18769.912,E2 -18769.912} C_VEL
LIN {X 0,Y 288.628,Z 342.532,A -85,B 0,C 180,E1 -18770.496,E2 -18770.496} C_VEL
LIN {X 0,Y 286.006,Z 357.556,A -85,B 0,C 180,E1 -18771.313,E2 -18771.313} C_VEL
LIN {X 0,Y 283.053,Z 371.087,A -85,B 0,C 180,E1 -18772.308,E2 -18772.308} C_VEL
LIN {X 0,Y 279.143,Z 386.08,A -85,B 0,C 180,E1 -18773.742,E2 -18773.742} C_VEL
LIN {X 0,Y 275.636,Z 398.029,A -85,B 0,C 180,E1 -18775.215,E2 -18775.215} C_VEL
LIN {X 0,Y 271.37,Z 410.433,A -85,B 0,C 180,E1 -18777.054,E2 -18777.054} C_VEL
LIN {X 0,Y 267.129,Z 421.755,A -85,B 0,C 180,E1 -18779.134,E2 -18779.134} C_VEL
LIN {X 0,Y 263.231,Z 431.33,A -85,B 0,C 180,E1 -18781.277,E2 -18781.277} C_VEL
LIN {X 0,Y 259.523,Z 440.27,A -85,B 0,C 180,E1 -18783.717,E2 -18783.717} C_VEL
LIN {X 0,Y 255.932,Z 448.674,A -85,B 0,C 180,E1 -18786.536,E2 -18786.536} C_VEL
LIN {X 0,Y 252.78,Z 456.097,A -85,B 0,C 180,E1 -18789.664,E2 -18789.664} C_VEL
LIN {X 0,Y 250.353,Z 461.718,A -85,B 0,C 180,E1 -18792.641,E2 -18792.641} C_VEL
LIN {X 0,Y 248.97,Z 465.593,A -85,B 0,C 180,E1 -18795.283,E2 -18795.283} C_VEL
LIN {X 0,Y 247.686,Z 469.27,A -85,B 0,C 180,E1 -18798.544,E2 -18798.544} C_VEL
LIN {X 0,Y 247.033,Z 471.776,A -85,B 0,C 180,E1 -18801.823,E2 -18801.823} C_VEL
LIN {X 0,Y 246.839,Z 473.15,A -85,B 0,C 180,E1 -18805.212,E2 -18805.212} C_VEL
LIN {X 0,Y 246.918,Z 473.295,A -85,B 0,C 180,E1 -18808.37,E2 -18808.37} C_VEL
LIN {X 0,Y 246.982,Z 472.959,A -85,B 0,C 180,E1 -18810.001,E2 -18810.001} C_VEL
LIN {X 0,Y 246.879,Z 471.408,A -85,B 0,C 180,E1 -18813.265,E2 -18813.265} C_VEL
LIN {X 0,Y 246.957,Z 468.656,A -85,B 0,C 180,E1 -18816.537,E2 -18816.537} C_VEL
LIN {X 0,Y 247.264,Z 464.621,A -85,B 0,C 180,E1 -18819.82,E2 -18819.82} C_VEL
LIN {X 0,Y 248.015,Z 459.181,A -85,B 0,C 180,E1 -18823.103,E2 -18823.103} C_VEL
LIN {X 0,Y 249.259,Z 452.202,A -85,B 0,C 180,E1 -18826.378,E2 -18826.378} C_VEL
LIN {X 0,Y 250.955,Z 444.663,A -85,B 0,C 180,E1 -18829.212,E2 -18829.212} C_VEL
LIN {X 0,Y 253.213,Z 435.596,A -85,B 0,C 180,E1 -18832.006,E2 -18832.006} C_VEL
LIN {X 0,Y 255.741,Z 425.19,A -85,B 0,C 180,E1 -18834.637,E2 -18834.637} C_VEL
LIN {X 0,Y 258.122,Z 415.342,A -85,B 0,C 180,E1 -18836.697,E2 -18836.697} C_VEL
LIN {X 0,Y 260.943,Z 403.348,A -85,B 0,C 180,E1 -18838.78,E2 -18838.78} C_VEL
LIN {X 0,Y 263.484,Z 391.652,A -85,B 0,C 180,E1 -18840.451,E2 -18840.451} C_VEL
LIN {X 0,Y 266.16,Z 378.221,A -85,B 0,C 180,E1 -18842.005,E2 -18842.005} C_VEL
LIN {X 0,Y 268.585,Z 363.686,A -85,B 0,C 180,E1 -18843.334,E2 -18843.334} C_VEL
LIN {X 0,Y 270.476,Z 349.919,A -85,B 0,C 180,E1 -18844.301,E2 -18844.301} C_VEL
LIN {X 0,Y 272.134,Z 334.502,A -85,B 0,C 180,E1 -18845.074,E2 -18845.074} C_VEL
LIN {X 0,Y 273.181,Z 318.301,A -85,B 0,C 180,E1 -18845.597,E2 -18845.597} C_VEL
LIN {X 0,Y 277.228,Z 221.87,A -85,B 0,C 180,E1 -18848.052,E2 -18848.052} C_VEL
LIN {X 0,Y 276.162,Z 215.897,A -85,B 0,C 180,E1 -18848.378,E2 -18848.378} C_VEL
LIN {X 0,Y 268.434,Z 196.882,A -85,B 0,C 180,E1 -18850.043,E2 -18850.043} C_VEL
LIN {X 0,Y 260.792,Z 180.222,A -85,B 0,C 180,E1 -18851.744,E2 -18851.744} C_VEL
LIN {X 0,Y 253.024,Z 165.202,A -85,B 0,C 180,E1 -18853.541,E2 -18853.541} C_VEL
LIN {X 0,Y 250.591,Z 160.585,A -85,B 0,C 180,E1 -18854.179,E2 -18854.179} C_VEL
LIN {X 0,Y 249.006,Z 155.098,A -85,B 0,C 180,E1 -18856.381,E2 -18856.381} C_VEL
LIN {X 0,Y 249.009,Z 155.088,A -85,B 0,C 180,E1 -18859.646,E2 -18859.646} C_VEL
LIN {X 0,Y 249.05,Z 155.086,A -85,B 0,C 180,E1 -18863.659,E2 -18863.659} C_VEL
LIN {X 0,Y 249.035,Z 155.086,A -85,B 0,C 180,E1 -18867.848,E2 -18867.848} C_VEL
LIN {X 0,Y 249.051,Z 155.059,A -85,B 0,C 180,E1 -18871.333,E2 -18871.333} C_VEL
LIN {X 0,Y 249.105,Z 155.071,A -85,B 0,C 180,E1 -18874.964,E2 -18874.964} C_VEL
LIN {X 0,Y 249.092,Z 155.071,A -85,B 0,C 180,E1 -18878.606,E2 -18878.606} C_VEL
LIN {X 0,Y 249.199,Z 155.06,A -85,B 0,C 180,E1 -18883.62,E2 -18883.62} C_VEL
LIN {X 0,Y 249.238,Z 155.058,A -85,B 0,C 180,E1 -18888.617,E2 -18888.617} C_VEL
LIN {X 0,Y 249.422,Z 155.034,A -85,B 0,C 180,E1 -18891.902,E2 -18891.902} C_VEL
LIN {X 0,Y 249.267,Z 155.058,A -85,B 0,C 180,E1 -18895.149,E2 -18895.149} C_VEL
LIN {X 0,Y 249.661,Z 154.974,A -85,B 0,C 180,E1 -18898.388,E2 -18898.388} C_VEL
LIN {X 0,Y 249.659,Z 154.988,A -85,B 0,C 180,E1 -18901.614,E2 -18901.614} C_VEL
LIN {X 0,Y 249.425,Z 155.027,A -85,B 0,C 180,E1 -18906.55,E2 -18906.55} C_VEL
LIN {X 0,Y 249.337,Z 155.007,A -85,B 0,C 180,E1 -18909.737,E2 -18909.737} C_VEL
LIN {X 0,Y 249.146,Z 155.073,A -85,B 0,C 180,E1 -18914.708,E2 -18914.708} C_VEL
LIN {X 0,Y 249.075,Z 155.078,A -85,B 0,C 180,E1 -18918.083,E2 -18918.083} C_VEL
LIN {X 0,Y 249.045,Z 155.079,A -85,B 0,C 180,E1 -18921.523,E2 -18921.523} C_VEL
LIN {X 0,Y 249.048,Z 155.085,A -85,B 0,C 180,E1 -18925.44,E2 -18925.44} C_VEL
LIN {X 0,Y 249.028,Z 155.05,A -85,B 0,C 180,E1 -18928.968,E2 -18928.968} C_VEL
LIN {X 0,Y 249.03,Z 155.082,A -85,B 0,C 180,E1 -18932.427,E2 -18932.427} C_VEL
LIN {X 0,Y 249.018,Z 155.071,A -85,B 0,C 180,E1 -18936.348,E2 -18936.348} C_VEL
LIN {X 0,Y 248.989,Z 155.083,A -85,B 0,C 180,E1 -18940.482,E2 -18940.482} C_VEL
LIN {X 0,Y 248.989,Z 155.094,A -85,B 0,C 180,E1 -18942.786,E2 -18942.786} C_VEL
LIN {X 0,Y 248.982,Z 155.078,A -85,B 0,C 180,E1 -18947.354,E2 -18947.354} C_VEL
LIN {X 0,Y 249.007,Z 155.075,A -85,B 0,C 180,E1 -18951.615,E2 -18951.615} C_VEL
LIN {X 0,Y 249.048,Z 155.087,A -85,B 0,C 180,E1 -18955.639,E2 -18955.639} C_VEL
LIN {X 0,Y 249.007,Z 155.096,A -85,B 0,C 180,E1 -18959.466,E2 -18959.466} C_VEL
LIN {X 0,Y 249.032,Z 155.091,A -85,B 0,C 180,E1 -18963.157,E2 -18963.157} C_VEL
LIN {X 0,Y 249.102,Z 155.251,A -85,B 0,C 180,E1 -18964.882,E2 -18964.882} C_VEL
LIN {X 0,Y 250.115,Z 158.02,A -85,B 0,C 180,E1 -18965.165,E2 -18965.165} C_VEL
LIN {X 0,Y 251.714,Z 160.235,A -85,B 0,C 180,E1 -18965.527,E2 -18965.527} C_VEL
LIN {X 0,Y 262.459,Z 178.051,A -85,B 0,C 180,E1 -18967.911,E2 -18967.911} C_VEL
LIN {X 0,Y 268.533,Z 189.549,A -85,B 0,C 180,E1 -18969.205,E2 -18969.205} C_VEL
LIN {X 0,Y 276.105,Z 207.191,A -85,B 0,C 180,E1 -18970.816,E2 -18970.816} C_VEL
LIN {X 0,Y 277.542,Z 210.732,A -85,B 0,C 180,E1 -18971.116,E2 -18971.116} C_VEL
LIN {X 0,Y 272.972,Z 314.802,A -85,B 0,C 180,E1 -18973.788,E2 -18973.788} C_VEL
LIN {X 0,Y 271.67,Z 330.58,A -85,B 0,C 180,E1 -18974.478,E2 -18974.478} C_VEL
LIN {X 0,Y 270.032,Z 345.071,A -85,B 0,C 180,E1 -18975.396,E2 -18975.396} C_VEL
LIN {X 0,Y 267.971,Z 358.982,A -85,B 0,C 180,E1 -18976.557,E2 -18976.557} C_VEL
LIN {X 0,Y 265.636,Z 372.326,A -85,B 0,C 180,E1 -18977.974,E2 -18977.974} C_VEL
LIN {X 0,Y 262.822,Z 386.117,A -85,B 0,C 180,E1 -18979.795,E2 -18979.795} C_VEL
LIN {X 0,Y 259.968,Z 398.59,A -85,B 0,C 180,E1 -18981.84,E2 -18981.84} C_VEL
LIN {X 0,Y 257.265,Z 409.917,A -85,B 0,C 180,E1 -18984.119,E2 -18984.119} C_VEL
LIN {X 0,Y 254.475,Z 420.962,A -85,B 0,C 180,E1 -18986.833,E2 -18986.833} C_VEL
LIN {X 0,Y 252.253,Z 429.972,A -85,B 0,C 180,E1 -18989.56,E2 -18989.56} C_VEL
LIN {X 0,Y 250.358,Z 437.691,A -85,B 0,C 180,E1 -18992.413,E2 -18992.413} C_VEL
LIN {X 0,Y 248.81,Z 444.791,A -85,B 0,C 180,E1 -18995.673,E2 -18995.673} C_VEL
LIN {X 0,Y 247.729,Z 450.378,A -85,B 0,C 180,E1 -18998.976,E2 -18998.976} C_VEL
LIN {X 0,Y 247.142,Z 453.668,A -85,B 0,C 180,E1 -19001.481,E2 -19001.481} C_VEL
LIN {X 0,Y 246.69,Z 456.932,A -85,B 0,C 180,E1 -19004.856,E2 -19004.856} C_VEL
LIN {X 0,Y 246.566,Z 458.942,A -85,B 0,C 180,E1 -19008.272,E2 -19008.272} C_VEL
LIN {X 0,Y 246.643,Z 459.688,A -85,B 0,C 180,E1 -19011.742,E2 -19011.742} C_VEL
LIN {X 0,Y 247.072,Z 459.153,A -85,B 0,C 180,E1 -19015.256,E2 -19015.256} C_VEL
LIN {X 0,Y 247.977,Z 457.3,A -85,B 0,C 180,E1 -19018.803,E2 -19018.803} C_VEL
LIN {X 0,Y 249.431,Z 454.049,A -85,B 0,C 180,E1 -19022.367,E2 -19022.367} C_VEL
LIN {X 0,Y 251.598,Z 449.299,A -85,B 0,C 180,E1 -19025.916,E2 -19025.916} C_VEL
LIN {X 0,Y 254.52,Z 442.914,A -85,B 0,C 180,E1 -19029.426,E2 -19029.426} C_VEL
LIN {X 0,Y 257.147,Z 437.134,A -85,B 0,C 180,E1 -19031.908,E2 -19031.908} C_VEL
LIN {X 0,Y 260.962,Z 428.453,A -85,B 0,C 180,E1 -19034.934,E2 -19034.934} C_VEL
LIN {X 0,Y 264.784,Z 419.482,A -85,B 0,C 180,E1 -19037.438,E2 -19037.438} C_VEL
LIN {X 0,Y 269.018,Z 408.915,A -85,B 0,C 180,E1 -19039.83,E2 -19039.83} C_VEL
LIN {X 0,Y 272.994,Z 398.048,A -85,B 0,C 180,E1 -19041.839,E2 -19041.839} C_VEL
LIN {X 0,Y 277.025,Z 385.976,A -85,B 0,C 180,E1 -19043.656,E2 -19043.656} C_VEL
LIN {X 0,Y 280.78,Z 373.252,A -85,B 0,C 180,E1 -19045.205,E2 -19045.205} C_VEL
LIN {X 0,Y 283.957,Z 360.328,A -85,B 0,C 180,E1 -19046.488,E2 -19046.488} C_VEL
LIN {X 0,Y 286.991,Z 345.674,A -85,B 0,C 180,E1 -19047.604,E2 -19047.604} C_VEL
LIN {X 0,Y 289.009,Z 333.127,A -85,B 0,C 180,E1 -19048.333,E2 -19048.333} C_VEL
LIN {X 0,Y 290.834,Z 317.999,A -85,B 0,C 180,E1 -19048.965,E2 -19048.965} C_VEL
LIN {X 0,Y 292.373,Z 294.723,A -85,B 0,C 180,E1 -19049.588,E2 -19049.588} C_VEL
LIN {X 0,Y 296.541,Z 224.67,A -85,B 0,C 180,E1 -19051.267,E2 -19051.267} C_VEL
LIN {X 0,Y 291.156,Z 213.873,A -85,B 0,C 180,E1 -19052.91,E2 -19052.91} C_VEL
LIN {X 0,Y 285.683,Z 204.052,A -85,B 0,C 180,E1 -19054.661,E2 -19054.661} C_VEL
LIN {X 0,Y 279.651,Z 194.124,A -85,B 0,C 180,E1 -19056.755,E2 -19056.755} C_VEL
LIN {X 0,Y 273.331,Z 185.404,A -85,B 0,C 180,E1 -19059.12,E2 -19059.12} C_VEL
